KUKA KRL program: MyProgram_105().src

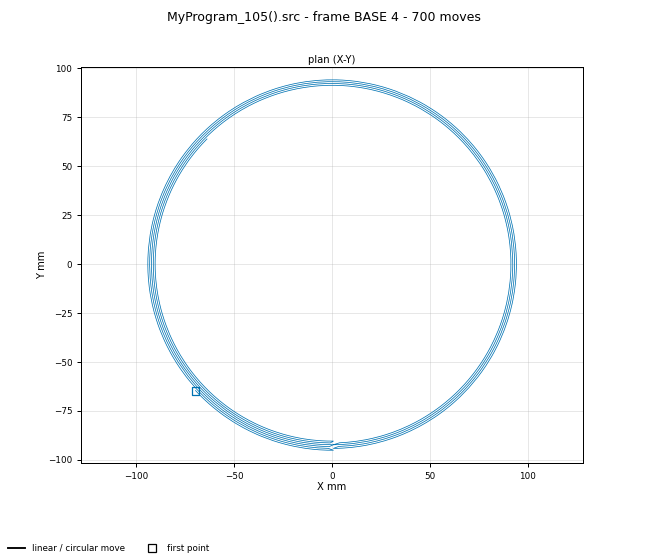
[picture p0: tool path of MyProgram_105().src in frame BASE 4, 700 of 700 moves have a stored position in this frame; points joined in program order, loops and branches not executed]
&ACCESS RVP
&REL 1
&PARAM TEMPLATE = C:\KRC\Roboter\Template\vorgabe
&PARAM EDITMASK = *
DEF MyProgram_105()
; ---- Setting reference (Base) ----
$BASE = BASE_DATA[4]

; --------------------------
; ---- Setting tool (TCP) ----
$TOOL = TOOL_DATA[3]
; --------------------------

$VEL.CP = VEL_APROX_PRINT
Startdeposition()
$VEL.CP = VEL_PRINT
LIN {X -69.7387,Y -64.5804,Z 94,A -141.1238,B 24.9322,C -1.9014,E1 24.8838,E2 -133.6356} C_DIS
LIN {X -67.3874,Y -67.0297,Z 94,A -139.0772,B 24.9325,C -1.897,E1 24.8878,E2 -135.6805} C_DIS
LIN {X -65.0404,Y -69.3086,Z 94,A -137.2267,B 24.9331,C -1.889,E1 24.8915,E2 -137.5194} C_DIS
LIN {X -62.8875,Y -71.2694,Z 94,A -135.3657,B 24.9331,C -1.889,E1 24.8954,E2 -139.3879} C_DIS
LIN {X -60.7875,Y -73.0672,Z 94,A -133.451,B 24.9327,C -1.8942,E1 24.8995,E2 -141.3222} C_DIS
LIN {X -57.6296,Y -75.5844,Z 94,A -131.3715,B 24.9339,C -1.8779,E1 24.904,E2 -143.3707} C_DIS
LIN {X -55.0629,Y -77.4728,Z 94,A -129.4404,B 24.9341,C -1.875,E1 24.9084,E2 -145.3015} C_DIS
LIN {X -51.0894,Y -80.1492,Z 94,A -126.4299,B 24.9341,C -1.8745,E1 24.9154,E2 -148.3208} C_DIS
LIN {X -49.1486,Y -81.3536,Z 94,A -124.3043,B 24.9325,C -1.898,E1 24.9207,E2 -150.5088} C_DIS
LIN {X -45.3379,Y -83.5369,Z 94,A -122.4556,B 24.9347,C -1.8671,E1 24.925,E2 -152.2894} C_DIS
LIN {X -42.3193,Y -85.1059,Z 94,A -120.7349,B 24.9356,C -1.8533,E1 24.9292,E2 -153.982} C_DIS
LIN {X -38.4134,Y -86.94,Z 94,A -117.9508,B 24.9354,C -1.8565,E1 24.9363,E2 -156.7806} C_DIS
LIN {X -36.0603,Y -87.9411,Z 94,A -116.4717,B 24.9357,C -1.8528,E1 24.9401,E2 -158.2542} C_DIS
LIN {X -30.1003,Y -90.1553,Z 94,A -112.2316,B 24.9349,C -1.8634,E1 24.9513,E2 -162.528} C_DIS
LIN {X -27.0209,Y -91.1252,Z 94,A -110.0331,B 24.9344,C -1.8708,E1 24.9573,E2 -164.7478} C_DIS
LIN {X -23.4233,Y -92.1159,Z 94,A -107.9464,B 24.9349,C -1.8638,E1 24.9629,E2 -166.8209} C_DIS
LIN {X -19.3908,Y -93.0484,Z 94,A -105.6833,B 24.9355,C -1.8545,E1 24.969,E2 -169.0649} C_DIS
LIN {X -13.8438,Y -94.0346,Z 94,A -102.1719,B 24.9353,C -1.8575,E1 24.9787,E2 -172.5866} C_DIS
LIN {X -9.7635,Y -94.5443,Z 94,A -99.8234,B 24.9357,C -1.8525,E1 24.9852,E2 -174.9249} C_DIS
LIN {X -6.5432,Y -94.8216,Z 94,A -97.8434,B 24.9356,C -1.8536,E1 24.9907,E2 -176.9083} C_DIS
LIN {X -2.4896,Y -95.0153,Z 94,A -95.2226,B 24.9351,C -1.8601,E1 24.998,E2 -179.5449} C_DIS
LIN {X 0.6469,Y -95.0437,Z 94,A -94.1191,B 24.937,C -1.8326,E1 25.0009,E2 -180.5833} C_DIS
Enddeposition()
LIN {X 0.6469,Y -95.0437,Z 94,A -94.1191,B 24.937,C -1.8326,E1 25.0009,E2 -180.5833} C_DIS
Startdeposition()
$VEL.CP = VEL_PRINT
LIN {X -1.9482,Y -94.0929,Z 94,A -96.3275,B 24.9374,C -1.8269,E1 24.9947,E2 -178.3611} C_DIS
LIN {X -6.9643,Y -93.8563,Z 94,A -99.1666,B 24.9369,C -1.8342,E1 24.9869,E2 -175.5385} C_DIS
LIN {X -11.9151,Y -93.3557,Z 94,A -101.987,B 24.9364,C -1.8417,E1 24.9791,E2 -172.7344} C_DIS
LIN {X -17.66,Y -92.4411,Z 94,A -105.2821,B 24.9358,C -1.8512,E1 24.9701,E2 -169.4586} C_DIS
LIN {X -22.5057,Y -91.3824,Z 94,A -108.5122,B 24.9362,C -1.8454,E1 24.9612,E2 -166.2106} C_DIS
LIN {X -25.5822,Y -90.5692,Z 94,A -110.5603,B 24.9363,C -1.8428,E1 24.9557,E2 -164.1533} C_DIS
LIN {X -28.6869,Y -89.6346,Z 94,A -113.2651,B 24.9379,C -1.8199,E1 24.9483,E2 -161.3892} C_DIS
LIN {X -32.4293,Y -88.3493,Z 94,A -115.1165,B 24.9365,C -1.8405,E1 24.9436,E2 -159.5831} C_DIS
LIN {X -35.4663,Y -87.1743,Z 94,A -117.1104,B 24.9364,C -1.842,E1 24.9384,E2 -157.5885} C_DIS
LIN {X -37.9827,Y -86.1086,Z 94,A -119.61,B 24.9382,C -1.8163,E1 24.9319,E2 -155.0218} C_DIS
LIN {X -42.4578,Y -83.9924,Z 94,A -121.6687,B 24.9358,C -1.8513,E1 24.9269,E2 -153.0409} C_DIS
LIN {X -48.2351,Y -80.8131,Z 94,A -125.5484,B 24.9351,C -1.8612,E1 24.9175,E2 -149.1735} C_DIS
LIN {X -50.3789,Y -79.4952,Z 94,A -128.169,B 24.9374,C -1.8282,E1 24.9111,E2 -146.4659} C_DIS
LIN {X -54.3758,Y -76.8154,Z 94,A -129.9375,B 24.9344,C -1.8706,E1 24.9072,E2 -144.7923} C_DIS
LIN {X -57.3626,Y -74.6107,Z 94,A -133.1316,B 24.9362,C -1.8443,E1 24.8999,E2 -141.5242} C_DIS
LIN {X -60.5001,Y -72.0913,Z 94,A -134.99,B 24.9346,C -1.8679,E1 24.8961,E2 -139.7148} C_DIS
LIN {X -62.7074,Y -70.1784,Z 94,A -136.6439,B 24.9341,C -1.8754,E1 24.8926,E2 -138.0722} C_DIS
LIN {X -64.8399,Y -68.2148,Z 94,A -138.555,B 24.9341,C -1.8742,E1 24.8887,E2 -136.1506} C_DIS
LIN {X -67.2732,Y -65.816,Z 94,A -140.6427,B 24.9339,C -1.8784,E1 24.8846,E2 -134.064} C_DIS
LIN {X -69.6416,Y -63.3045,Z 94,A -142.8737,B 24.9339,C -1.8789,E1 24.8803,E2 -131.8244} C_DIS
LIN {X -73.0499,Y -59.3376,Z 94,A -145.4867,B 24.932,C -1.9045,E1 24.8757,E2 -129.2603} C_DIS
LIN {X -74.6075,Y -57.3668,Z 94,A -148.2971,B 24.9346,C -1.8677,E1 24.8708,E2 -126.3489} C_DIS
LIN {X -77.3825,Y -53.5649,Z 94,A -149.7414,B 24.9309,C -1.9196,E1 24.8686,E2 -125.0212} C_DIS
LIN {X -79.2935,Y -50.6931,Z 94,A -153.1451,B 24.9335,C -1.8839,E1 24.8633,E2 -121.5154} C_DIS
LIN {X -81.4743,Y -47.1085,Z 94,A -154.6711,B 24.9307,C -1.9229,E1 24.8612,E2 -120.0743} C_DIS
LIN {X -82.5961,Y -45.113,Z 94,A -156.3966,B 24.9312,C -1.9162,E1 24.8588,E2 -118.3238} C_DIS
LIN {X -84.3717,Y -41.6972,Z 94,A -158.9654,B 24.9312,C -1.9156,E1 24.8556,E2 -115.7399} C_DIS
LIN {X -85.8006,Y -38.6713,Z 94,A -160.8303,B 24.9304,C -1.9267,E1 24.8534,E2 -113.8913} C_DIS
LIN {X -87.9215,Y -33.5723,Z 94,A -163.8897,B 24.929,C -1.9459,E1 24.8502,E2 -110.8606} C_DIS
LIN {X -88.9552,Y -30.7311,Z 94,A -166.0977,B 24.9295,C -1.9398,E1 24.8481,E2 -108.6256} C_DIS
LIN {X -89.9802,Y -27.5839,Z 94,A -168.0075,B 24.9288,C -1.9492,E1 24.8465,E2 -106.7271} C_DIS
LIN {X -90.8948,Y -24.4003,Z 94,A -170.161,B 24.9286,C -1.951,E1 24.8449,E2 -104.5656} C_DIS
LIN {X -91.8007,Y -20.7376,Z 94,A -172.5876,B 24.9284,C -1.9541,E1 24.8433,E2 -102.132} C_DIS
LIN {X -92.9269,Y -14.9027,Z 94,A -176.0707,B 24.9273,C -1.9695,E1 24.8416,E2 -98.665} C_DIS
LIN {X -93.3738,Y -11.7751,Z 94,A -178.7651,B 24.9286,C -1.952,E1 24.8406,E2 -95.9128} C_DIS
LIN {X -93.8172,Y -7.4536,Z 94,A 178.8539,B 24.9274,C -1.9684,E1 24.8401,E2 -93.5567} C_DIS
LIN {X -94.024,Y -4.0875,Z 94,A 177.0484,B 24.9263,C -1.9825,E1 24.8399,E2 -91.774} C_DIS
LIN {X -94.1117,Y -0.5106,Z 94,A 174.5652,B 24.9265,C -1.9802,E1 24.8399,E2 -89.2703} C_DIS
LIN {X -94.0669,Y 2.9403,Z 94,A 173.1792,B 24.9243,C -2.0088,E1 24.8399,E2 -87.9442} C_DIS
LIN {X -93.7885,Y 7.8127,Z 94,A 170.2835,B 24.9234,C -2.0207,E1 24.8404,E2 -85.0593} C_DIS
LIN {X -92.8908,Y 15.1219,Z 94,A 165.6955,B 24.9226,C -2.0318,E1 24.842,E2 -80.4705} C_DIS
LIN {X -91.9219,Y 20.189,Z 94,A 162.4209,B 24.9221,C -2.0376,E1 24.8438,E2 -77.1905} C_DIS
LIN {X -91.2356,Y 23.0956,Z 94,A 160.1751,B 24.9227,C -2.0303,E1 24.8453,E2 -74.914} C_DIS
LIN {X -90.0393,Y 27.3932,Z 94,A 157.4118,B 24.9222,C -2.0373,E1 24.8474,E2 -72.1515} C_DIS
LIN {X -88.776,Y 31.2417,Z 94,A 155.2063,B 24.921,C -2.053,E1 24.8494,E2 -69.9708} C_DIS
LIN {X -86.7799,Y 36.421,Z 94,A 151.5856,B 24.9207,C -2.0559,E1 24.8532,E2 -66.3368} C_DIS
LIN {X -85.0096,Y 40.3813,Z 94,A 148.9037,B 24.9202,C -2.0625,E1 24.8563,E2 -63.6561} C_DIS
LIN {X -82.7539,Y 44.822,Z 94,A 145.7368,B 24.9199,C -2.0673,E1 24.8604,E2 -60.4838} C_DIS
LIN {X -80.3279,Y 49.0375,Z 94,A 143.0972,B 24.9184,C -2.0857,E1 24.8641,E2 -57.8743} C_DIS
LIN {X -78.336,Y 52.162,Z 94,A 140.8604,B 24.9179,C -2.0926,E1 24.8675,E2 -55.6427} C_DIS
LIN {X -76.808,Y 54.3862,Z 94,A 139.1867,B 24.9176,C -2.0961,E1 24.8702,E2 -53.9692} C_DIS
LIN {X -74.738,Y 57.1974,Z 94,A 137.0233,B 24.9172,C -2.1006,E1 24.8739,E2 -51.8062} C_DIS
LIN {X -71.3643,Y 61.3558,Z 94,A 133.7903,B 24.9165,C -2.1099,E1 24.8796,E2 -48.5805} C_DIS
LIN {X -69.2025,Y 63.7831,Z 94,A 131.2365,B 24.9175,C -2.097,E1 24.8845,E2 -45.9845} C_DIS
LIN {X -66.5924,Y 66.5052,Z 94,A 128.9093,B 24.9172,C -2.1015,E1 24.8891,E2 -43.6583} C_DIS
LIN {X -63.895,Y 69.0998,Z 94,A 127.1979,B 24.9153,C -2.1246,E1 24.8925,E2 -41.9949} C_DIS
LIN {X -61.3973,Y 71.3289,Z 94,A 124.3388,B 24.917,C -2.1035,E1 24.8987,E2 -39.0743} C_DIS
LIN {X -57.8983,Y 74.195,Z 94,A 122.515,B 24.9142,C -2.1386,E1 24.9025,E2 -37.3273} C_DIS
LIN {X -55.5308,Y 75.9839,Z 94,A 120.6043,B 24.9142,C -2.139,E1 24.9068,E2 -35.4108} C_DIS
LIN {X -52.6421,Y 78.0131,Z 94,A 118.4191,B 24.9139,C -2.1421,E1 24.9118,E2 -33.2257} C_DIS
LIN {X -49.0591,Y 80.3148,Z 94,A 115.5451,B 24.9143,C -2.138,E1 24.9186,E2 -30.3328} C_DIS
LIN {X -45.2932,Y 82.4983,Z 94,A 112.9239,B 24.9138,C -2.1435,E1 24.925,E2 -27.7172} C_DIS
LIN {X -39.0636,Y 85.6239,Z 94,A 109.1301,B 24.9121,C -2.1647,E1 24.9344,E2 -23.9639} C_DIS
LIN {X -36.6843,Y 86.6689,Z 94,A 106.2784,B 24.9152,C -2.1262,E1 24.942,E2 -21.014} C_DIS
LIN {X -31.6825,Y 88.6205,Z 94,A 103.9563,B 24.9124,C -2.1609,E1 24.9479,E2 -18.7695} C_DIS
LIN {X -28.1024,Y 89.8194,Z 94,A 101.1148,B 24.9136,C -2.1459,E1 24.9555,E2 -15.8874} C_DIS
LIN {X -24.4026,Y 90.8942,Z 94,A 98.8913,B 24.9131,C -2.1523,E1 24.9615,E2 -13.6756} C_DIS
LIN {X -21.0964,Y 91.7179,Z 94,A 97.5058,B 24.9111,C -2.1768,E1 24.9651,E2 -12.3465} C_DIS
LIN {X -18.6315,Y 92.2506,Z 94,A 94.7987,B 24.9141,C -2.1396,E1 24.9728,E2 -9.5481} C_DIS
LIN {X -13.6027,Y 93.1253,Z 94,A 92.9169,B 24.9107,C -2.1821,E1 24.9777,E2 -7.7655} C_DIS
LIN {X -7.7308,Y 93.795,Z 94,A 89.1085,B 24.9111,C -2.177,E1 24.9883,E2 -3.9426} C_DIS
LIN {X -2.724,Y 94.0735,Z 94,A 86.0802,B 24.911,C -2.1789,E1 24.9967,E2 -0.918} C_DIS
LIN {X 2.2075,Y 94.0881,Z 94,A 83.1336,B 24.9108,C -2.1813,E1 25.005,E2 2.0227} C_DIS
LIN {X 5.2902,Y 93.964,Z 94,A 80.5365,B 24.9127,C -2.1571,E1 25.0124,E2 4.6762} C_DIS
LIN {X 9.0331,Y 93.6791,Z 94,A 79.1257,B 24.9103,C -2.1865,E1 25.0161,E2 6.0165} C_DIS
LIN {X 12.6316,Y 93.262,Z 94,A 76.4626,B 24.9116,C -2.1704,E1 25.0236,E2 8.7157} C_DIS
LIN {X 19.2709,Y 92.1193,Z 94,A 72.6653,B 24.9109,C -2.1793,E1 25.0339,E2 12.4877} C_DIS
LIN {X 22.378,Y 91.4136,Z 94,A 70.5662,B 24.9115,C -2.1728,E1 25.0397,E2 14.5994} C_DIS
LIN {X 25.7736,Y 90.5149,Z 94,A 67.8851,B 24.9131,C -2.1526,E1 25.047,E2 17.3237} C_DIS
LIN {X 29.3297,Y 89.4266,Z 94,A 66.1402,B 24.9118,C -2.1687,E1 25.0515,E2 19.0272} C_DIS
LIN {X 32.4829,Y 88.3297,Z 94,A 63.9325,B 24.9124,C -2.1608,E1 25.0574,E2 21.2491} C_DIS
LIN {X 39.4143,Y 85.4625,Z 94,A 59.7402,B 24.9118,C -2.169,E1 25.0681,E2 25.4121} C_DIS
LIN {X 44.9057,Y 82.7085,Z 94,A 56.0161,B 24.9121,C -2.1648,E1 25.0773,E2 29.1359} C_DIS
LIN {X 47.5693,Y 81.2066,Z 94,A 53.309,B 24.9147,C -2.1323,E1 25.084,E2 31.9119} C_DIS
LIN {X 51.1467,Y 79.0023,Z 94,A 51.6246,B 24.9126,C -2.1592,E1 25.0878,E2 33.5271} C_DIS
LIN {X 53.4154,Y 77.4865,Z 94,A 49.8003,B 24.9132,C -2.1507,E1 25.0921,E2 35.3654} C_DIS
LIN {X 55.8489,Y 75.751,Z 94,A 47.9869,B 24.9135,C -2.1478,E1 25.0962,E2 37.1794} C_DIS
LIN {X 57.8006,Y 74.2732,Z 94,A 46.327,B 24.9142,C -2.139,E1 25.0999,E2 38.8539} C_DIS
LIN {X 60.7815,Y 71.8535,Z 94,A 44.2061,B 24.9139,C -2.1423,E1 25.1044,E2 40.9588} C_DIS
LIN {X 63.4363,Y 69.5206,Z 94,A 41.9455,B 24.9146,C -2.1341,E1 25.1091,E2 43.2297} C_DIS
LIN {X 65.4276,Y 67.6496,Z 94,A 40.3764,B 24.9146,C -2.1341,E1 25.1123,E2 44.7924} C_DIS
LIN {X 69.153,Y 63.8368,Z 94,A 36.8128,B 24.9161,C -2.1155,E1 25.1192,E2 48.3845} C_DIS
LIN {X 72.2885,Y 60.2629,Z 94,A 34.2832,B 24.9155,C -2.1221,E1 25.1237,E2 50.8871} C_DIS
LIN {X 74.6663,Y 57.2905,Z 94,A 31.7816,B 24.9165,C -2.1098,E1 25.1281,E2 53.4059} C_DIS
LIN {X 76.8074,Y 54.3871,Z 94,A 29.7489,B 24.9165,C -2.1103,E1 25.1314,E2 55.4276} C_DIS
LIN {X 78.7198,Y 51.5799,Z 94,A 27.6645,B 24.9169,C -2.1044,E1 25.1346,E2 57.5155} C_DIS
LIN {X 80.6364,Y 48.53,Z 94,A 25.3599,B 24.9177,C -2.0945,E1 25.138,E2 59.8317} C_DIS
LIN {X 83.4996,Y 43.4198,Z 94,A 21.9255,B 24.9181,C -2.0897,E1 25.1426,E2 63.2596} C_DIS
LIN {X 85.0801,Y 40.2357,Z 94,A 19.7798,B 24.9185,C -2.0843,E1 25.1452,E2 65.4064} C_DIS
LIN {X 87.3911,Y 34.9333,Z 94,A 16.2834,B 24.9192,C -2.0751,E1 25.149,E2 68.9054} C_DIS
LIN {X 88.6183,Y 31.6912,Z 94,A 13.6184,B 24.9213,C -2.0484,E1 25.1516,E2 71.6186} C_DIS
LIN {X 89.8436,Y 28.0226,Z 94,A 11.6623,B 24.9207,C -2.0561,E1 25.1532,E2 73.5454} C_DIS
LIN {X 90.732,Y 25.0029,Z 94,A 9.6745,B 24.9214,C -2.0476,E1 25.1547,E2 75.5418} C_DIS
LIN {X 92.0604,Y 19.5543,Z 94,A 5.9044,B 24.9232,C -2.0238,E1 25.157,E2 79.3461} C_DIS
LIN {X 92.8381,Y 15.4375,Z 94,A 4.0615,B 24.9218,C -2.0422,E1 25.1579,E2 81.1348} C_DIS
LIN {X 93.6449,Y 9.3822,Z 94,A 0.5547,B 24.9221,C -2.0384,E1 25.1591,E2 84.6299} C_DIS
LIN {X 93.9475,Y 5.5898,Z 94,A -1.9705,B 24.9232,C -2.0232,E1 25.1596,E2 87.176} C_DIS
LIN {X 94.0861,Y 2.3126,Z 94,A -3.9319,B 24.9236,C -2.0181,E1 25.1598,E2 89.1378} C_DIS
LIN {X 94.0913,Y -2.0333,Z 94,A -6.8642,B 24.9251,C -1.9989,E1 25.1597,E2 92.098} C_DIS
LIN {X 93.8432,Y -7.1286,Z 94,A -9.5757,B 24.9247,C -2.0036,E1 25.1592,E2 94.7822} C_DIS
LIN {X 93.551,Y -10.2794,Z 94,A -12.0195,B 24.9266,C -1.978,E1 25.1585,E2 97.2719} C_DIS
LIN {X 93.103,Y -13.7597,Z 94,A -13.4432,B 24.9252,C -1.9979,E1 25.158,E2 98.6403} C_DIS
LIN {X 92.3502,Y -18.1321,Z 94,A -16.1344,B 24.9258,C -1.9896,E1 25.1567,E2 101.3353} C_DIS
LIN {X 91.8924,Y -20.3244,Z 94,A -17.7291,B 24.9268,C -1.9766,E1 25.1557,E2 102.9515} C_DIS
LIN {X 91.0157,Y -23.9512,Z 94,A -19.9981,B 24.9273,C -1.9694,E1 25.1541,E2 105.2242} C_DIS
LIN {X 89.6895,Y -28.5172,Z 94,A -22.8587,B 24.9279,C -1.9616,E1 25.1518,E2 108.0869} C_DIS
LIN {X 87.8435,Y -33.7781,Z 94,A -26.1921,B 24.9285,C -1.9534,E1 25.1487,E2 111.421} C_DIS
LIN {X 85.7242,Y -38.8408,Z 94,A -29.3311,B 24.9286,C -1.9509,E1 25.1453,E2 114.5489} C_DIS
LIN {X 84.517,Y -41.404,Z 94,A -31.2668,B 24.9296,C -1.9378,E1 25.1429,E2 116.5051} C_DIS
LIN {X 82.6594,Y -44.9962,Z 94,A -33.4527,B 24.9294,C -1.9409,E1 25.1401,E2 118.6721} C_DIS
LIN {X 81.4822,Y -47.0949,Z 94,A -35.2037,B 24.9305,C -1.9259,E1 25.1376,E2 120.4494} C_DIS
LIN {X 78.5782,Y -51.7946,Z 94,A -38.347,B 24.9305,C -1.9246,E1 25.1329,E2 123.5799} C_DIS
LIN {X 76.3889,Y -54.9736,Z 94,A -40.547,B 24.9306,C -1.9237,E1 25.1294,E2 125.7712} C_DIS
LIN {X 74.3614,Y -57.6861,Z 94,A -43.1709,B 24.9325,C -1.8972,E1 25.1249,E2 128.4451} C_DIS
LIN {X 69.8011,Y -63.1288,Z 94,A -46.9332,B 24.9318,C -1.9068,E1 25.1182,E2 132.1677} C_DIS
LIN {X 65.1773,Y -67.8909,Z 94,A -51.8243,B 24.9348,C -1.8657,E1 25.1084,E2 137.1352} C_DIS
LIN {X 62.1685,Y -70.6571,Z 94,A -53.4027,B 24.9328,C -1.8933,E1 25.1052,E2 138.6421} C_DIS
LIN {X 60.1046,Y -72.42,Z 94,A -55.9394,B 24.9353,C -1.8572,E1 25.0996,E2 141.2541} C_DIS
LIN {X 56.8954,Y -74.969,Z 94,A -58.1928,B 24.9351,C -1.8607,E1 25.0947,E2 143.4913} C_DIS
LIN {X 54.2953,Y -76.8729,Z 94,A -59.6964,B 24.9342,C -1.8733,E1 25.0913,E2 144.9597} C_DIS
LIN {X 52.3467,Y -78.2132,Z 94,A -62.078,B 24.9368,C -1.8364,E1 25.0856,E2 147.4207} C_DIS
LIN {X 48.145,Y -80.8664,Z 94,A -64.5264,B 24.9357,C -1.8515,E1 25.0799,E2 149.8258} C_DIS
LIN {X 44.3104,Y -83.0305,Z 94,A -67.7405,B 24.9374,C -1.8278,E1 25.0718,E2 153.0868} C_DIS
LIN {X 39.9429,Y -85.2164,Z 94,A -70.5367,B 24.9373,C -1.8294,E1 25.0648,E2 155.872} C_DIS
LIN {X 35.9424,Y -86.9805,Z 94,A -72.4829,B 24.9358,C -1.851,E1 25.0599,E2 157.7624} C_DIS
LIN {X 32.7951,Y -88.2157,Z 94,A -74.6569,B 24.9363,C -1.8441,E1 25.0542,E2 159.9481} C_DIS
LIN {X 30.2093,Y -89.1327,Z 94,A -76.2525,B 24.9363,C -1.8447,E1 25.05,E2 161.5392} C_DIS
LIN {X 26.5766,Y -90.2825,Z 94,A -79.3116,B 24.9382,C -1.8159,E1 25.0417,E2 164.6611} C_DIS
LIN {X 22.086,Y -91.4849,Z 94,A -80.9658,B 24.9355,C -1.8546,E1 25.0375,E2 166.2213} C_DIS
LIN {X 17.5884,Y -92.4549,Z 94,A -84.0246,B 24.9363,C -1.8429,E1 25.029,E2 169.3038} C_DIS
LIN {X 14.3248,Y -93.0162,Z 94,A -86.79,B 24.9382,C -1.8152,E1 25.0212,E2 172.1321} C_DIS
LIN {X 10.2227,Y -93.5569,Z 94,A -88.3941,B 24.9362,C -1.8456,E1 25.017,E2 173.663} C_DIS
LIN {X 5.4967,Y -93.9526,Z 94,A -91.2131,B 24.9361,C -1.8466,E1 25.0092,E2 176.4783} C_DIS
LIN {X 2.829,Y -94.0703,Z 94,A -93.0455,B 24.9366,C -1.8388,E1 25.004,E2 178.3286} C_DIS
LIN {X 0.6498,Y -94.1008,Z 94,A -94.5174,B 24.937,C -1.8335,E1 24.9998,E2 179.8128} C_DIS
Enddeposition()
LIN {X 0.6498,Y -94.1008,Z 94,A -94.5174,B 24.937,C -1.8335,E1 24.9998,E2 179.8128} C_DIS
Startdeposition()
$VEL.CP = VEL_PRINT
LIN {X 3.2914,Y -93.1215,Z 94,A -91.9183,B 24.9335,C -1.8841,E1 25.0074,E2 177.0944} C_DIS
LIN {X 10.2483,Y -92.6149,Z 94,A -87.8414,B 24.9338,C -1.8786,E1 25.0187,E2 173.0324} C_DIS
LIN {X 15.9916,Y -91.7975,Z 94,A -84.2081,B 24.9335,C -1.8834,E1 25.0288,E2 169.3912} C_DIS
LIN {X 18.5909,Y -91.3053,Z 94,A -82.0498,B 24.9321,C -1.9037,E1 25.0348,E2 167.1873} C_DIS
LIN {X 22.9029,Y -90.3203,Z 94,A -79.1877,B 24.9315,C -1.9115,E1 25.0426,E2 164.3109} C_DIS
LIN {X 26.3762,Y -89.3676,Z 94,A -77.5356,B 24.9328,C -1.8938,E1 25.0469,E2 162.7037} C_DIS
LIN {X 29.7303,Y -88.3083,Z 94,A -75.4252,B 24.9328,C -1.8945,E1 25.0525,E2 160.5955} C_DIS
LIN {X 33.1365,Y -87.0876,Z 94,A -73.0879,B 24.9322,C -1.9015,E1 25.0587,E2 158.2466} C_DIS
LIN {X 35.6068,Y -86.1085,Z 94,A -71.1636,B 24.9313,C -1.9144,E1 25.0637,E2 156.2963} C_DIS
LIN {X 39.7153,Y -84.292,Z 94,A -68.8745,B 24.9322,C -1.9014,E1 25.0694,E2 154.0435} C_DIS
LIN {X 44.1269,Y -82.0682,Z 94,A -65.6924,B 24.9315,C -1.9117,E1 25.0774,E2 150.8458} C_DIS
LIN {X 47.7244,Y -80.0298,Z 94,A -62.6462,B 24.9298,C -1.9349,E1 25.0848,E2 147.7543} C_DIS
LIN {X 50.8647,Y -78.0724,Z 94,A -60.8908,B 24.9309,C -1.9201,E1 25.0888,E2 146.0395} C_DIS
LIN {X 53.7993,Y -76.0792,Z 94,A -58.2456,B 24.9293,C -1.9417,E1 25.095,E2 143.3524} C_DIS
LIN {X 56.6324,Y -73.994,Z 94,A -56.446,B 24.93,C -1.9328,E1 25.0989,E2 141.5804} C_DIS
LIN {X 60.6404,Y -70.7465,Z 94,A -53.6631,B 24.9305,C -1.9255,E1 25.1049,E2 138.8254} C_DIS
LIN {X 63.0794,Y -68.5803,Z 94,A -51.3646,B 24.9294,C -1.9409,E1 25.1097,E2 136.4995} C_DIS
LIN {X 65.8763,Y -65.8989,Z 94,A -48.9558,B 24.9289,C -1.9477,E1 25.1145,E2 134.085} C_DIS
LIN {X 68.5042,Y -63.1624,Z 94,A -46.333,B 24.9277,C -1.9643,E1 25.1195,E2 131.4343} C_DIS
LIN {X 72.2287,Y -58.8671,Z 94,A -43.2821,B 24.9282,C -1.9568,E1 25.125,E2 128.4153} C_DIS
LIN {X 74.8639,Y -55.4791,Z 94,A -40.618,B 24.9276,C -1.9648,E1 25.1295,E2 125.7449} C_DIS
LIN {X 76.6192,Y -53.0263,Z 94,A -38.5078,B 24.9265,C -1.9795,E1 25.1329,E2 123.6102} C_DIS
LIN {X 80.2312,Y -47.3837,Z 94,A -34.8052,B 24.9268,C -1.9755,E1 25.1383,E2 119.9358} C_DIS
LIN {X 81.8823,Y -44.4695,Z 94,A -32.7879,B 24.9265,C -1.9799,E1 25.1411,E2 117.9186} C_DIS
LIN {X 83.4573,Y -41.4383,Z 94,A -30.6607,B 24.926,C -1.9872,E1 25.1438,E2 115.7856} C_DIS
LIN {X 84.7648,Y -38.6962,Z 94,A -28.1751,B 24.9238,C -2.0161,E1 25.1467,E2 113.2451} C_DIS
LIN {X 86.217,Y -35.3404,Z 94,A -26.5433,B 24.925,C -1.9996,E1 25.1484,E2 111.6612} C_DIS
LIN {X 88.2401,Y -29.9328,Z 94,A -23.0282,B 24.9243,C -2.0092,E1 25.1518,E2 108.1431} C_DIS
LIN {X 89.0893,Y -27.3028,Z 94,A -21.1469,B 24.9234,C -2.0214,E1 25.1534,E2 106.2437} C_DIS
LIN {X 90.3026,Y -22.9726,Z 94,A -18.5312,B 24.9231,C -2.0245,E1 25.1552,E2 103.6358} C_DIS
LIN {X 91.095,Y -19.5966,Z 94,A -15.3708,B 24.9196,C -2.0706,E1 25.1572,E2 100.3852} C_DIS
LIN {X 92.0816,Y -14.2557,Z 94,A -13.5788,B 24.9233,C -2.0223,E1 25.1579,E2 98.7175} C_DIS
LIN {X 92.7097,Y -9.3435,Z 94,A -10.0316,B 24.9211,C -2.051,E1 25.1592,E2 95.1236} C_DIS
LIN {X 92.9685,Y -6.2546,Z 94,A -7.5808,B 24.919,C -2.0779,E1 25.1596,E2 92.6239} C_DIS
LIN {X 93.1514,Y -2.3147,Z 94,A -5.3074,B 24.9189,C -2.0798,E1 25.1598,E2 90.3595} C_DIS
LIN {X 93.1739,Y 1.0661,Z 94,A -3.6792,B 24.9197,C -2.0694,E1 25.1598,E2 88.7656} C_DIS
LIN {X 93.0629,Y 4.6669,Z 94,A -0.9336,B 24.9176,C -2.0966,E1 25.1594,E2 85.972} C_DIS
LIN {X 92.8008,Y 8.3839,Z 94,A 0.3782,B 24.9199,C -2.0668,E1 25.1591,E2 84.7383} C_DIS
LIN {X 92.0264,Y 14.6133,Z 94,A 4.1664,B 24.9192,C -2.0762,E1 25.1578,E2 80.9503} C_DIS
LIN {X 91.485,Y 17.6848,Z 94,A 6.6821,B 24.9169,C -2.1047,E1 25.1565,E2 78.3821} C_DIS
LIN {X 90.6237,Y 21.6696,Z 94,A 9.1578,B 24.9164,C -2.1112,E1 25.1549,E2 75.9053} C_DIS
LIN {X 89.6254,Y 25.4862,Z 94,A 11.2153,B 24.9169,C -2.1048,E1 25.1535,E2 73.8748} C_DIS
LIN {X 87.5444,Y 31.9098,Z 94,A 15.4946,B 24.9156,C -2.1218,E1 25.1497,E2 69.5795} C_DIS
LIN {X 86.383,Y 34.9324,Z 94,A 17.777,B 24.9142,C -2.1385,E1 25.1473,E2 67.2703} C_DIS
LIN {X 84.2155,Y 39.8783,Z 94,A 20.6943,B 24.9147,C -2.1329,E1 25.144,E2 64.3822} C_DIS
LIN {X 81.9335,Y 44.3747,Z 94,A 24.4268,B 24.9121,C -2.165,E1 25.1391,E2 60.5936} C_DIS
LIN {X 80.1355,Y 47.5455,Z 94,A 26.1711,B 24.9131,C -2.1524,E1 25.1366,E2 58.888} C_DIS
LIN {X 78.3117,Y 50.4933,Z 94,A 28.3066,B 24.9126,C -2.1581,E1 25.1334,E2 56.7498} C_DIS
LIN {X 76.212,Y 53.6121,Z 94,A 30.3869,B 24.9129,C -2.1554,E1 25.1302,E2 54.6862} C_DIS
LIN {X 74.5248,Y 55.9313,Z 94,A 32.8088,B 24.9105,C -2.1841,E1 25.126,E2 52.2081} C_DIS
LIN {X 72.334,Y 58.7371,Z 94,A 34.5233,B 24.9115,C -2.1717,E1 25.1231,E2 50.5308} C_DIS
LIN {X 70.0892,Y 61.3985,Z 94,A 37.4122,B 24.9089,C -2.2042,E1 25.1177,E2 47.578} C_DIS
LIN {X 66.9704,Y 64.7862,Z 94,A 39.4361,B 24.9108,C -2.1806,E1 25.1139,E2 45.6187} C_DIS
LIN {X 64.5539,Y 67.1943,Z 94,A 41.456,B 24.9107,C -2.1822,E1 25.1099,E2 43.6035} C_DIS
LIN {X 60.9408,Y 70.489,Z 94,A 44.5547,B 24.9099,C -2.1915,E1 25.1034,E2 40.4952} C_DIS
LIN {X 59.052,Y 72.0788,Z 94,A 46.125,B 24.9095,C -2.1962,E1 25.1,E2 38.9197} C_DIS
LIN {X 56.5971,Y 74.0213,Z 94,A 48.1948,B 24.9088,C -2.205,E1 25.0954,E2 36.8369} C_DIS
LIN {X 52.9441,Y 76.6763,Z 94,A 50.6792,B 24.9093,C -2.1991,E1 25.0898,E2 34.3749} C_DIS
LIN {X 48.4077,Y 79.6174,Z 94,A 54.0116,B 24.9088,C -2.2045,E1 25.0819,E2 31.0405} C_DIS
LIN {X 45.3335,Y 81.4072,Z 94,A 55.8988,B 24.9095,C -2.197,E1 25.0774,E2 29.1769} C_DIS
LIN {X 39.8714,Y 84.2188,Z 94,A 59.9732,B 24.9082,C -2.2122,E1 25.0672,E2 25.0775} C_DIS
LIN {X 34.5103,Y 86.5536,Z 94,A 63.6897,B 24.9075,C -2.2203,E1 25.0576,E2 21.3506} C_DIS
LIN {X 30.9656,Y 87.8829,Z 94,A 65.6061,B 24.9086,C -2.208,E1 25.0527,E2 19.4674} C_DIS
LIN {X 26.0415,Y 89.4669,Z 94,A 69.0272,B 24.9077,C -2.2188,E1 25.0435,E2 16.0269} C_DIS
LIN {X 23.0761,Y 90.276,Z 94,A 70.857,B 24.9077,C -2.2179,E1 25.0386,E2 14.2021} C_DIS
LIN {X 20.7277,Y 90.8442,Z 94,A 72.5671,B 24.907,C -2.2264,E1 25.0339,E2 12.474} C_DIS
LIN {X 15.1554,Y 91.9381,Z 94,A 75.9548,B 24.9072,C -2.2242,E1 25.0246,E2 9.0955} C_DIS
LIN {X 8.6612,Y 92.7752,Z 94,A 79.575,B 24.9083,C -2.211,E1 25.0147,E2 5.5093} C_DIS
LIN {X 3.6923,Y 93.1059,Z 94,A 82.8341,B 24.9077,C -2.2176,E1 25.0056,E2 2.2358} C_DIS
LIN {X -2.0956,Y 93.1558,Z 94,A 86.7375,B 24.9068,C -2.2286,E1 24.9946,E2 -1.6934} C_DIS
LIN {X -7.6443,Y 92.8648,Z 94,A 89.6946,B 24.9082,C -2.2118,E1 24.9865,E2 -4.6116} C_DIS
LIN {X -13.835,Y 92.1467,Z 94,A 93.5529,B 24.9084,C -2.2103,E1 24.9758,E2 -8.4691} C_DIS
LIN {X -19.2391,Y 91.1722,Z 94,A 97.2689,B 24.9076,C -2.2189,E1 24.9655,E2 -12.2094} C_DIS
LIN {X -21.8619,Y 90.5779,Z 94,A 99.7551,B 24.9054,C -2.2451,E1 24.9586,E2 -14.7614} C_DIS
LIN {X -26.5767,Y 89.3081,Z 94,A 101.8119,B 24.9083,C -2.2104,E1 24.9533,E2 -16.7391} C_DIS
LIN {X -29.7671,Y 88.2959,Z 94,A 103.6106,B 24.9093,C -2.1995,E1 24.9485,E2 -18.5151} C_DIS
LIN {X -33.957,Y 86.7709,Z 94,A 107.2306,B 24.9072,C -2.2247,E1 24.9389,E2 -22.2025} C_DIS
LIN {X -37.3474,Y 85.3665,Z 94,A 108.8945,B 24.909,C -2.202,E1 24.9348,E2 -23.8164} C_DIS
LIN {X -42.6543,Y 82.8429,Z 94,A 112.9932,B 24.9082,C -2.212,E1 24.9244,E2 -27.9497} C_DIS
LIN {X -46.7524,Y 80.6015,Z 94,A 115.487,B 24.9096,C -2.1947,E1 24.9184,E2 -30.4095} C_DIS
LIN {X -49.8777,Y 78.7068,Z 94,A 117.8468,B 24.9096,C -2.1941,E1 24.9128,E2 -32.7754} C_DIS
LIN {X -53.2048,Y 76.4951,Z 94,A 120.1566,B 24.9105,C -2.1846,E1 24.9075,E2 -35.0703} C_DIS
LIN {X -56.1183,Y 74.3843,Z 94,A 123.3638,B 24.9082,C -2.2121,E1 24.9002,E2 -38.3544} C_DIS
LIN {X -60.1304,Y 71.181,Z 94,A 125.5502,B 24.9114,C -2.1739,E1 24.8957,E2 -40.4582} C_DIS
LIN {X -62.598,Y 69.022,Z 94,A 127.6474,B 24.9115,C -2.1719,E1 24.8913,E2 -42.5589} C_DIS
LIN {X -66.1153,Y 65.6588,Z 94,A 130.9478,B 24.9113,C -2.1745,E1 24.8847,E2 -45.8795} C_DIS
LIN {X -69.3234,Y 62.2619,Z 94,A 133.4609,B 24.9128,C -2.156,E1 24.88,E2 -48.3594} C_DIS
LIN {X -71.3342,Y 59.9495,Z 94,A 136.0473,B 24.9114,C -2.1733,E1 24.8753,E2 -50.999} C_DIS
LIN {X -73.8181,Y 56.8608,Z 94,A 137.7695,B 24.9138,C -2.1443,E1 24.8724,E2 -52.6601} C_DIS
LIN {X -75.8326,Y 54.1449,Z 94,A 139.8967,B 24.9141,C -2.1402,E1 24.8689,E2 -54.7878} C_DIS
LIN {X -77.3263,Y 51.9902,Z 94,A 141.6584,B 24.9141,C -2.1404,E1 24.8661,E2 -56.5588} C_DIS
LIN {X -79.3802,Y 48.7982,Z 94,A 143.9166,B 24.9148,C -2.1314,E1 24.8628,E2 -58.807} C_DIS
LIN {X -82.2505,Y 43.7868,Z 94,A 147.4953,B 24.9156,C -2.122,E1 24.8579,E2 -62.382} C_DIS
LIN {X -84.6675,Y 38.9085,Z 94,A 150.8241,B 24.9164,C -2.1114,E1 24.8539,E2 -65.7037} C_DIS
LIN {X -85.7078,Y 36.5595,Z 94,A 153.2367,B 24.9147,C -2.1326,E1 24.8512,E2 -68.1802} C_DIS
LIN {X -87.3826,Y 32.3533,Z 94,A 155.2484,B 24.9173,C -2.1,E1 24.8493,E2 -70.1253} C_DIS
LIN {X -88.3047,Y 29.7411,Z 94,A 157.1625,B 24.9172,C -2.1012,E1 24.8475,E2 -72.0534} C_DIS
LIN {X -89.6428,Y 25.4247,Z 94,A 159.7005,B 24.9185,C -2.0851,E1 24.8455,E2 -74.5674} C_DIS
LIN {X -90.5207,Y 22.0964,Z 94,A 161.7975,B 24.919,C -2.0778,E1 24.8441,E2 -76.6593} C_DIS
LIN {X -91.1619,Y 19.2891,Z 94,A 164.2361,B 24.9179,C -2.0929,E1 24.8426,E2 -79.1482} C_DIS
LIN {X -91.8473,Y 15.6985,Z 94,A 165.6303,B 24.9205,C -2.0593,E1 24.842,E2 -80.4705} C_DIS
LIN {X -92.5284,Y 10.9893,Z 94,A 168.8462,B 24.9205,C -2.0588,E1 24.8408,E2 -83.7044} C_DIS
LIN {X -92.8693,Y 7.5875,Z 94,A 170.8247,B 24.9213,C -2.0482,E1 24.8402,E2 -85.6696} C_DIS
LIN {X -93.1159,Y 3.4561,Z 94,A 174.3057,B 24.9197,C -2.0691,E1 24.8398,E2 -89.2214} C_DIS
LIN {X -93.1755,Y -0.8477,Z 94,A 176.0725,B 24.9225,C -2.0333,E1 24.8398,E2 -90.9133} C_DIS
LIN {X -92.9273,Y -6.8625,Z 94,A 179.782,B 24.9234,C -2.0216,E1 24.8403,E2 -94.6173} C_DIS
LIN {X -92.5083,Y -11.1615,Z 94,A -177.362,B 24.9235,C -2.0194,E1 24.8411,E2 -97.4852} C_DIS
LIN {X -92.0422,Y -14.5106,Z 94,A -175.3181,B 24.9241,C -2.0118,E1 24.842,E2 -99.523} C_DIS
LIN {X -91.1752,Y -19.224,Z 94,A -172.2501,B 24.9245,C -2.0064,E1 24.8436,E2 -102.5962} C_DIS
LIN {X -90.4415,Y -22.421,Z 94,A -170.2426,B 24.925,C -1.9999,E1 24.8449,E2 -104.6001} C_DIS
LIN {X -89.5464,Y -25.7651,Z 94,A -168.1255,B 24.9255,C -1.9931,E1 24.8465,E2 -106.7132} C_DIS
LIN {X -88.5253,Y -29.0808,Z 94,A -166.1584,B 24.9264,C -1.9815,E1 24.8481,E2 -108.664} C_DIS
LIN {X -87.8315,Y -31.112,Z 94,A -164.5745,B 24.9261,C -1.9859,E1 24.8496,E2 -110.2673} C_DIS
LIN {X -86.3446,Y -35.0267,Z 94,A -161.7799,B 24.9261,C -1.9853,E1 24.8525,E2 -113.0762} C_DIS
LIN {X -84.5217,Y -39.2217,Z 94,A -159.4756,B 24.9279,C -1.9614,E1 24.8551,E2 -115.336} C_DIS
LIN {X -82.5612,Y -43.1969,Z 94,A -156.5373,B 24.9279,C -1.9605,E1 24.8588,E2 -118.288} C_DIS
LIN {X -80.9968,Y -46.0646,Z 94,A -154.7322,B 24.9288,C -1.9486,E1 24.8612,E2 -120.0743} C_DIS
LIN {X -78.4931,Y -50.2106,Z 94,A -151.3534,B 24.9285,C -1.9535,E1 24.8662,E2 -123.4821} C_DIS
LIN {X -73.5996,Y -57.1443,Z 94,A -146.2415,B 24.9296,C -1.9371,E1 24.8745,E2 -128.5798} C_DIS
LIN {X -70.1694,Y -61.3067,Z 94,A -142.9473,B 24.9303,C -1.9287,E1 24.8804,E2 -131.8691} C_DIS
LIN {X -67.857,Y -63.8567,Z 94,A -140.8395,B 24.9306,C -1.9238,E1 24.8844,E2 -133.9743} C_DIS
LIN {X -65.4928,Y -66.2793,Z 94,A -138.7695,B 24.931,C -1.919,E1 24.8885,E2 -136.0417} C_DIS
LIN {X -63.1472,Y -68.518,Z 94,A -136.6394,B 24.931,C -1.9193,E1 24.8928,E2 -138.1814} C_DIS
LIN {X -60.2117,Y -71.1118,Z 94,A -133.1597,B 24.9287,C -1.9499,E1 24.9004,E2 -141.7474} C_DIS
LIN {X -55.862,Y -74.5768,Z 94,A -130.9791,B 24.9321,C -1.903,E1 24.905,E2 -143.8242} C_DIS
LIN {X -52.1729,Y -77.2027,Z 94,A -127.635,B 24.9311,C -1.9168,E1 24.9128,E2 -147.2126} C_DIS
LIN {X -48.2625,Y -79.7058,Z 94,A -125.3392,B 24.9327,C -1.894,E1 24.9181,E2 -149.4614} C_DIS
LIN {X -43.0441,Y -82.6416,Z 94,A -121.4825,B 24.9327,C -1.8948,E1 24.9276,E2 -153.3309} C_DIS
LIN {X -40.6817,Y -83.8295,Z 94,A -119.3485,B 24.9316,C -1.9098,E1 24.9331,E2 -155.5063} C_DIS
LIN {X -37.552,Y -85.2773,Z 94,A -117.5842,B 24.9326,C -1.8955,E1 24.9375,E2 -157.2409} C_DIS
LIN {X -33.9039,Y -86.7918,Z 94,A -115.6356,B 24.934,C -1.877,E1 24.9424,E2 -159.1498} C_DIS
LIN {X -29.3053,Y -88.4517,Z 94,A -112.2664,B 24.9333,C -1.8866,E1 24.9514,E2 -162.5484} C_DIS
LIN {X -26.0544,Y -89.463,Z 94,A -110.1257,B 24.9333,C -1.8867,E1 24.9571,E2 -164.693} C_DIS
LIN {X -21.768,Y -90.6008,Z 94,A -106.8808,B 24.9321,C -1.903,E1 24.966,E2 -167.981} C_DIS
LIN {X -18.1192,Y -91.4014,Z 94,A -105.113,B 24.9335,C -1.8838,E1 24.9707,E2 -169.7053} C_DIS
LIN {X -14.0135,Y -92.1191,Z 94,A -102.4496,B 24.9333,C -1.8865,E1 24.9781,E2 -172.3777} C_DIS
LIN {X -7.6203,Y -92.8667,Z 94,A -98.6745,B 24.9338,C -1.8797,E1 24.9885,E2 -176.1389} C_DIS
LIN {X -5.0764,Y -93.0402,Z 94,A -96.503,B 24.9323,C -1.9008,E1 24.9947,E2 -178.3612} C_DIS
LIN {X -1.4057,Y -93.1685,Z 94,A -93.9531,B 24.9315,C -1.9115,E1 25.0019,E2 -180.9365} C_DIS
LIN {X -1.4057,Y -93.1685,Z 94,A -93.9531,B 24.9315,C -1.9115,E1 25.0019,E2 -180.9365} C_DIS
Enddeposition()
LIN {X 0.6403,Y -92.241,Z 94,A -94.4274,B 24.9346,C -1.8679,E1 25.0003,E2 -180.3586} C_DIS
Startdeposition()
$VEL.CP = VEL_PRINT
LIN {X -5.4551,Y -92.0837,Z 94,A -98.1404,B 24.9345,C -1.8698,E1 24.99,E2 -176.6497} C_DIS
LIN {X -9.6737,Y -91.7358,Z 94,A -100.9603,B 24.9349,C -1.8636,E1 24.9821,E2 -173.8136} C_DIS
LIN {X -14.6853,Y -91.0695,Z 94,A -103.9212,B 24.9344,C -1.8702,E1 24.9739,E2 -170.8661} C_DIS
LIN {X -17.1169,Y -90.643,Z 94,A -105.5917,B 24.9347,C -1.8662,E1 24.9693,E2 -169.1843} C_DIS
LIN {X -21.0274,Y -89.8162,Z 94,A -108.0991,B 24.9347,C -1.8665,E1 24.9625,E2 -166.6746} C_DIS
LIN {X -23.4635,Y -89.2119,Z 94,A -109.7752,B 24.9349,C -1.8636,E1 24.9579,E2 -164.9889} C_DIS
LIN {X -26.9203,Y -88.2298,Z 94,A -111.8822,B 24.9345,C -1.8692,E1 24.9523,E2 -162.8919} C_DIS
LIN {X -29.6817,Y -87.3389,Z 94,A -114.0532,B 24.9352,C -1.8586,E1 24.9465,E2 -160.6917} C_DIS
LIN {X -33.9357,Y -85.7756,Z 94,A -116.7043,B 24.9347,C -1.8666,E1 24.9396,E2 -158.0538} C_DIS
LIN {X -36.885,Y -84.549,Z 94,A -118.6667,B 24.9345,C -1.8694,E1 24.9345,E2 -156.0936} C_DIS
LIN {X -40.1192,Y -83.0633,Z 94,A -120.7361,B 24.934,C -1.8765,E1 24.9293,E2 -154.0359} C_DIS
LIN {X -43.4315,Y -81.3818,Z 94,A -123.5549,B 24.9349,C -1.8631,E1 24.9223,E2 -151.1773} C_DIS
LIN {X -46.3995,Y -79.7269,Z 94,A -125.0185,B 24.9333,C -1.8867,E1 24.9189,E2 -149.7656} C_DIS
LIN {X -48.8455,Y -78.2506,Z 94,A -128.246,B 24.9363,C -1.8435,E1 24.911,E2 -146.4251} C_DIS
LIN {X -53.9752,Y -74.8061,Z 94,A -130.6054,B 24.9326,C -1.8963,E1 24.9059,E2 -144.1833} C_DIS
LIN {X -59.9227,Y -70.1307,Z 94,A -135.4052,B 24.9322,C -1.9017,E1 24.8953,E2 -139.3785} C_DIS
LIN {X -62.028,Y -68.2772,Z 94,A -137.3614,B 24.9324,C -1.8984,E1 24.8912,E2 -137.4065} C_DIS
LIN {X -64.6496,Y -65.7991,Z 94,A -139.5328,B 24.932,C -1.9052,E1 24.8869,E2 -135.2423} C_DIS
LIN {X -67.0104,Y -63.3933,Z 94,A -141.6028,B 24.9316,C -1.9104,E1 24.8829,E2 -133.1759} C_DIS
LIN {X -69.2653,Y -60.9217,Z 94,A -143.7073,B 24.9313,C -1.9142,E1 24.879,E2 -131.0711} C_DIS
LIN {X -71.8044,Y -57.9069,Z 94,A -146.0439,B 24.9306,C -1.9234,E1 24.8748,E2 -128.7456} C_DIS
LIN {X -75.4331,Y -53.0959,Z 94,A -149.9944,B 24.9305,C -1.9261,E1 24.8682,E2 -124.7824} C_DIS
LIN {X -77.2515,Y -50.4125,Z 94,A -152.766,B 24.9317,C -1.9081,E1 24.8639,E2 -121.9541} C_DIS
LIN {X -79.5698,Y -46.6667,Z 94,A -154.5361,B 24.9291,C -1.9448,E1 24.8615,E2 -120.2623} C_DIS
LIN {X -80.8806,Y -44.357,Z 94,A -156.3977,B 24.9292,C -1.9427,E1 24.8589,E2 -118.386} C_DIS
LIN {X -82.7927,Y -40.6757,Z 94,A -158.7596,B 24.9282,C -1.9564,E1 24.8559,E2 -116.044} C_DIS
LIN {X -83.917,Y -38.3037,Z 94,A -160.6006,B 24.9284,C -1.9545,E1 24.8538,E2 -114.1886} C_DIS
LIN {X -86.136,Y -33.0115,Z 94,A -163.928,B 24.9271,C -1.972,E1 24.8503,E2 -110.8843} C_DIS
LIN {X -87.3858,Y -29.5426,Z 94,A -166.0646,B 24.9262,C -1.9834,E1 24.8482,E2 -108.7629} C_DIS
LIN {X -88.5058,Y -25.9965,Z 94,A -168.8124,B 24.9267,C -1.977,E1 24.8459,E2 -105.9841} C_DIS
LIN {X -89.4071,Y -22.704,Z 94,A -170.934,B 24.9262,C -1.9835,E1 24.8444,E2 -103.8654} C_DIS
LIN {X -90.1719,Y -19.445,Z 94,A -173.1432,B 24.9261,C -1.986,E1 24.8431,E2 -101.6491} C_DIS
LIN {X -90.8971,Y -15.7167,Z 94,A -175.5155,B 24.9255,C -1.9929,E1 24.8419,E2 -99.2794} C_DIS
LIN {X -91.4489,Y -12.0912,Z 94,A -177.74,B 24.9249,C -2.0017,E1 24.841,E2 -97.0626} C_DIS
LIN {X -91.9186,Y -7.7568,Z 94,A 179.6488,B 24.924,C -2.0131,E1 24.8403,E2 -94.463} C_DIS
LIN {X -92.1889,Y -3.223,Z 94,A 176.7424,B 24.9235,C -2.0196,E1 24.8398,E2 -91.5545} C_DIS
LIN {X -92.2455,Y -0.0816,Z 94,A 174.301,B 24.9242,C -2.0112,E1 24.8398,E2 -89.0784} C_DIS
LIN {X -92.1044,Y 5.08,Z 94,A 171.5319,B 24.9224,C -2.0346,E1 24.8401,E2 -86.3485} C_DIS
LIN {X -91.8567,Y 8.4484,Z 94,A 169.3919,B 24.922,C -2.04,E1 24.8406,E2 -84.2087} C_DIS
LIN {X -91.4605,Y 12.0011,Z 94,A 166.8615,B 24.9221,C -2.0379,E1 24.8415,E2 -81.658} C_DIS
LIN {X -90.867,Y 15.888,Z 94,A 164.4276,B 24.9215,C -2.0459,E1 24.8426,E2 -79.2289} C_DIS
LIN {X -90.1424,Y 19.5802,Z 94,A 162.3666,B 24.9203,C -2.0616,E1 24.8437,E2 -77.1931} C_DIS
LIN {X -89.329,Y 23.0081,Z 94,A 160.2169,B 24.9197,C -2.0697,E1 24.8452,E2 -75.0501} C_DIS
LIN {X -88.5103,Y 25.9815,Z 94,A 157.541,B 24.921,C -2.0531,E1 24.8473,E2 -72.3191} C_DIS
LIN {X -87.3031,Y 29.7877,Z 94,A 155.6476,B 24.919,C -2.0782,E1 24.8489,E2 -70.4748} C_DIS
LIN {X -85.5086,Y 34.6027,Z 94,A 152.7188,B 24.9176,C -2.0959,E1 24.8518,E2 -67.5717} C_DIS
LIN {X -84.3659,Y 37.3049,Z 94,A 150.6129,B 24.9179,C -2.0928,E1 24.8542,E2 -65.4469} C_DIS
LIN {X -81.9398,Y 42.3681,Z 94,A 147.3378,B 24.9165,C -2.1096,E1 24.8582,E2 -62.1941} C_DIS
LIN {X -80.892,Y 44.3361,Z 94,A 145.2658,B 24.9179,C -2.093,E1 24.861,E2 -60.0715} C_DIS
LIN {X -79.2152,Y 47.2667,Z 94,A 143.8105,B 24.9158,C -2.1182,E1 24.863,E2 -58.669} C_DIS
LIN {X -77.624,Y 49.8351,Z 94,A 141.7184,B 24.9159,C -2.117,E1 24.8661,E2 -56.5633} C_DIS
LIN {X -75.8362,Y 52.516,Z 94,A 139.7847,B 24.9153,C -2.1246,E1 24.8691,E2 -54.6381} C_DIS
LIN {X -73.9938,Y 55.0828,Z 94,A 137.7524,B 24.9151,C -2.1278,E1 24.8725,E2 -52.6036} C_DIS
LIN {X -71.3037,Y 58.5244,Z 94,A 135.2089,B 24.9141,C -2.1401,E1 24.8769,E2 -50.0775} C_DIS
LIN {X -69.4653,Y 60.6927,Z 94,A 133.3214,B 24.9141,C -2.1409,E1 24.8803,E2 -48.1833} C_DIS
LIN {X -67.1446,Y 63.2507,Z 94,A 130.967,B 24.9141,C -2.1399,E1 24.8848,E2 -45.8161} C_DIS
LIN {X -64.0427,Y 66.3895,Z 94,A 128.4022,B 24.9132,C -2.1518,E1 24.8899,E2 -43.2689} C_DIS
LIN {X -61.5893,Y 68.6716,Z 94,A 126.2879,B 24.9128,C -2.1556,E1 24.8942,E2 -41.1551} C_DIS
LIN {X -58.9559,Y 70.9453,Z 94,A 123.5558,B 24.9139,C -2.1429,E1 24.9001,E2 -38.3823} C_DIS
LIN {X -56.1978,Y 73.1496,Z 94,A 122.0931,B 24.9117,C -2.17,E1 24.9032,E2 -36.9788} C_DIS
LIN {X -54.0134,Y 74.7788,Z 94,A 120.1208,B 24.9121,C -2.1648,E1 24.9077,E2 -34.9871} C_DIS
LIN {X -51.1173,Y 76.7869,Z 94,A 117.9077,B 24.9118,C -2.1684,E1 24.9128,E2 -32.7751} C_DIS
LIN {X -48.7849,Y 78.2884,Z 94,A 116.3512,B 24.9111,C -2.1768,E1 24.9165,E2 -31.2337} C_DIS
LIN {X -46.4978,Y 79.6696,Z 94,A 114.7549,B 24.9107,C -2.1817,E1 24.9203,E2 -29.6444} C_DIS
LIN {X -42.1928,Y 82.0296,Z 94,A 111.6309,B 24.9105,C -2.1846,E1 24.928,E2 -26.5182} C_DIS
LIN {X -39.5593,Y 83.3324,Z 94,A 109.6422,B 24.9107,C -2.1823,E1 24.933,E2 -24.519} C_DIS
LIN {X -36.5791,Y 84.6823,Z 94,A 107.6768,B 24.9103,C -2.1874,E1 24.938,E2 -22.5609} C_DIS
LIN {X -30.5744,Y 87.0301,Z 94,A 103.8111,B 24.9095,C -2.1971,E1 24.948,E2 -18.7102} C_DIS
LIN {X -27.866,Y 87.9365,Z 94,A 101.1274,B 24.9117,C -2.1703,E1 24.9554,E2 -15.958} C_DIS
LIN {X -23.8665,Y 89.1037,Z 94,A 99.5025,B 24.9089,C -2.2036,E1 24.9595,E2 -14.4099} C_DIS
LIN {X -21.5054,Y 89.7033,Z 94,A 97.7876,B 24.9093,C -2.1986,E1 24.9642,E2 -12.6805} C_DIS
LIN {X -18.3169,Y 90.4079,Z 94,A 95.2459,B 24.9105,C -2.1838,E1 24.9713,E2 -10.1008} C_DIS
LIN {X -15.0508,Y 91.0084,Z 94,A 93.854,B 24.9086,C -2.207,E1 24.9749,E2 -8.7625} C_DIS
LIN {X -10.2553,Y 91.6738,Z 94,A 90.7594,B 24.9087,C -2.2059,E1 24.9835,E2 -5.6631} C_DIS
LIN {X -7.1027,Y 91.9709,Z 94,A 88.1015,B 24.9105,C -2.1844,E1 24.9911,E2 -2.9529} C_DIS
LIN {X -3.4352,Y 92.1808,Z 94,A 86.5589,B 24.9084,C -2.2093,E1 24.9952,E2 -1.469} C_DIS
LIN {X 2.0466,Y 92.2224,Z 94,A 83.2393,B 24.9082,C -2.2128,E1 25.0045,E2 1.8423} C_DIS
LIN {X 7.1606,Y 91.9663,Z 94,A 79.8674,B 24.9087,C -2.2064,E1 25.0139,E2 5.2279} C_DIS
LIN {X 11.6,Y 91.5125,Z 94,A 77.3697,B 24.908,C -2.2152,E1 25.0208,E2 7.7032} C_DIS
LIN {X 14.02,Y 91.1728,Z 94,A 75.5539,B 24.9088,C -2.2048,E1 25.0258,E2 9.542} C_DIS
LIN {X 17.7804,Y 90.5153,Z 94,A 73.1467,B 24.909,C -2.2026,E1 25.0325,E2 11.9516} C_DIS
LIN {X 20.2489,Y 89.9958,Z 94,A 71.6175,B 24.909,C -2.2031,E1 25.0366,E2 13.4776} C_DIS
LIN {X 23.2363,Y 89.2703,Z 94,A 69.6176,B 24.9093,C -2.1989,E1 25.0421,E2 15.4844} C_DIS
LIN {X 26.5988,Y 88.3271,Z 94,A 67.2114,B 24.9101,C -2.1894,E1 25.0486,E2 17.9091} C_DIS
LIN {X 30.7634,Y 86.9638,Z 94,A 64.6182,B 24.9099,C -2.1914,E1 25.0554,E2 20.4924} C_DIS
LIN {X 33.9246,Y 85.78,Z 94,A 62.3963,B 24.9104,C -2.1851,E1 25.0612,E2 22.7243} C_DIS
LIN {X 37.2905,Y 84.3722,Z 94,A 60.4203,B 24.9098,C -2.1925,E1 25.0662,E2 24.678} C_DIS
LIN {X 40.4902,Y 82.8846,Z 94,A 57.7345,B 24.9114,C -2.1729,E1 25.073,E2 27.4032} C_DIS
LIN {X 43.5739,Y 81.3054,Z 94,A 56.1785,B 24.91,C -2.1906,E1 25.0768,E2 28.913} C_DIS
LIN {X 46.1489,Y 79.8709,Z 94,A 53.2137,B 24.9134,C -2.149,E1 25.0842,E2 31.9673} C_DIS
LIN {X 50.7324,Y 77.0405,Z 94,A 51.0217,B 24.9106,C -2.1836,E1 25.0891,E2 34.0704} C_DIS
LIN {X 52.8633,Y 75.5948,Z 94,A 48.7379,B 24.9127,C -2.1571,E1 25.0944,E2 36.409} C_DIS
LIN {X 55.9732,Y 73.3227,Z 94,A 46.9148,B 24.9115,C -2.1726,E1 25.0984,E2 38.1886} C_DIS
LIN {X 58.7963,Y 71.0779,Z 94,A 44.7812,B 24.9115,C -2.1722,E1 25.103,E2 40.3152} C_DIS
LIN {X 61.6673,Y 68.6018,Z 94,A 42.6151,B 24.9113,C -2.1743,E1 25.1076,E2 42.4679} C_DIS
LIN {X 63.5117,Y 66.899,Z 94,A 40.789,B 24.9124,C -2.1616,E1 25.1113,E2 44.3164} C_DIS
LIN {X 65.8983,Y 64.5492,Z 94,A 38.7393,B 24.9126,C -2.1583,E1 25.1154,E2 46.3653} C_DIS
LIN {X 69.2649,Y 60.9222,Z 94,A 35.7236,B 24.913,C -2.1535,E1 25.121,E2 49.379} C_DIS
LIN {X 71.4583,Y 58.3339,Z 94,A 32.7218,B 24.916,C -2.1168,E1 25.1265,E2 52.4535} C_DIS
LIN {X 74.3816,Y 54.5565,Z 94,A 30.9098,B 24.9132,C -2.1507,E1 25.1294,E2 54.1769} C_DIS
LIN {X 75.8558,Y 52.4878,Z 94,A 29.0975,B 24.9142,C -2.1383,E1 25.1323,E2 56.0096} C_DIS
LIN {X 77.6799,Y 49.7482,Z 94,A 27.1403,B 24.9144,C -2.1362,E1 25.1353,E2 57.9621} C_DIS
LIN {X 79.4488,Y 46.8713,Z 94,A 24.5024,B 24.9164,C -2.1112,E1 25.1391,E2 60.6454} C_DIS
LIN {X 81.0902,Y 43.9707,Z 94,A 22.4658,B 24.9168,C -2.1068,E1 25.1418,E2 62.6818} C_DIS
LIN {X 82.5953,Y 41.074,Z 94,A 21.315,B 24.9147,C -2.1329,E1 25.1432,E2 63.7648} C_DIS
LIN {X 83.6224,Y 38.9402,Z 94,A 18.5782,B 24.9186,C -2.083,E1 25.1466,E2 66.6047} C_DIS
LIN {X 85.497,Y 34.6312,Z 94,A 16.4942,B 24.9169,C -2.1046,E1 25.1487,E2 68.626} C_DIS
LIN {X 86.7781,Y 31.2844,Z 94,A 13.6692,B 24.9191,C -2.0764,E1 25.1515,E2 71.5019} C_DIS
LIN {X 88.0422,Y 27.5254,Z 94,A 12.0203,B 24.9174,C -2.0986,E1 25.1528,E2 73.0891} C_DIS
LIN {X 88.8096,Y 24.9386,Z 94,A 10.1457,B 24.9184,C -2.0863,E1 25.1543,E2 74.9821} C_DIS
LIN {X 89.9649,Y 20.3839,Z 94,A 6.6796,B 24.9206,C -2.0574,E1 25.1566,E2 78.4962} C_DIS
LIN {X 90.743,Y 16.5773,Z 94,A 5.2545,B 24.9184,C -2.086,E1 25.1573,E2 79.8455} C_DIS
LIN {X 91.1654,Y 14.0675,Z 94,A 2.8863,B 24.921,C -2.0522,E1 25.1583,E2 82.2797} C_DIS
LIN {X 91.6105,Y 10.7959,Z 94,A 1.1375,B 24.9207,C -2.0567,E1 25.1589,E2 84.0074} C_DIS
LIN {X 92.1691,Y 3.7343,Z 94,A -2.4483,B 24.9194,C -2.0727,E1 25.1597,E2 87.5341} C_DIS
LIN {X 92.2411,Y -0.806,Z 94,A -5.8863,B 24.9219,C -2.0408,E1 25.1597,E2 91.0269} C_DIS
LIN {X 92.1205,Y -4.7669,Z 94,A -8.6117,B 24.9232,C -2.0232,E1 25.1594,E2 93.7777} C_DIS
LIN {X 91.8761,Y -8.2382,Z 94,A -11.6992,B 24.9263,C -1.9825,E1 25.1586,E2 96.9428} C_DIS
LIN {X 91.1389,Y -14.2395,Z 94,A -15.0596,B 24.9261,C -1.9848,E1 25.1572,E2 100.2781} C_DIS
LIN {X 90.2773,Y -18.9529,Z 94,A -17.1579,B 24.9244,C -2.0074,E1 25.1561,E2 102.311} C_DIS
LIN {X 88.8627,Y -24.7513,Z 94,A -20.7882,B 24.9251,C -1.9984,E1 25.1536,E2 105.9414} C_DIS
LIN {X 87.9235,Y -27.9062,Z 94,A -22.9319,B 24.9259,C -1.9884,E1 25.1518,E2 108.0966} C_DIS
LIN {X 86.3563,Y -32.4294,Z 94,A -25.8429,B 24.9264,C -1.9815,E1 25.1491,E2 111.0076} C_DIS
LIN {X 84.506,Y -36.9837,Z 94,A -28.8194,B 24.9269,C -1.975,E1 25.1459,E2 113.983} C_DIS
LIN {X 82.7704,Y -40.7207,Z 94,A -31.5794,B 24.928,C -1.96,E1 25.1425,E2 116.7636} C_DIS
LIN {X 80.9545,Y -44.2208,Z 94,A -33.7691,B 24.9278,C -1.9623,E1 25.1397,E2 118.9363} C_DIS
LIN {X 79.3805,Y -46.9869,Z 94,A -36.0712,B 24.9291,C -1.9447,E1 25.1364,E2 121.2681} C_DIS
LIN {X 76.8576,Y -51.0099,Z 94,A -38.6456,B 24.9287,C -1.95,E1 25.1326,E2 123.8169} C_DIS
LIN {X 74.9656,Y -53.7516,Z 94,A -40.8053,B 24.9294,C -1.941,E1 25.1291,E2 125.9874} C_DIS
LIN {X 72.0153,Y -57.6454,Z 94,A -44.4566,B 24.9316,C -1.9106,E1 25.1227,E2 129.6933} C_DIS
LIN {X 69.4443,Y -60.7167,Z 94,A -46.1158,B 24.9299,C -1.9341,E1 25.1198,E2 131.2894} C_DIS
LIN {X 67.4197,Y -62.9581,Z 94,A -48.7703,B 24.9322,C -1.9013,E1 25.1146,E2 134.0097} C_DIS
LIN {X 64.6717,Y -65.7773,Z 94,A -50.5226,B 24.9309,C -1.9203,E1 25.1113,E2 135.7098} C_DIS
LIN {X 61.9722,Y -68.3284,Z 94,A -52.8835,B 24.9314,C -1.9129,E1 25.1064,E2 138.0785} C_DIS
LIN {X 59.426,Y -70.5539,Z 94,A -55.5021,B 24.9331,C -1.8897,E1 25.1008,E2 140.742} C_DIS
LIN {X 56.6132,Y -72.8295,Z 94,A -57.3793,B 24.9325,C -1.898,E1 25.0967,E2 142.5925} C_DIS
LIN {X 53.8372,Y -74.9045,Z 94,A -59.3253,B 24.9323,C -1.9009,E1 25.0923,E2 144.5247} C_DIS
LIN {X 50.9808,Y -76.8768,Z 94,A -61.4747,B 24.9325,C -1.8969,E1 25.0873,E2 146.6764} C_DIS
LIN {X 47.3039,Y -79.1932,Z 94,A -64.1414,B 24.9328,C -1.8929,E1 25.081,E2 149.344} C_DIS
LIN {X 45.3159,Y -80.3471,Z 94,A -65.5705,B 24.933,C -1.8903,E1 25.0775,E2 150.775} C_DIS
LIN {X 41.5819,Y -82.3411,Z 94,A -68.3566,B 24.9337,C -1.8803,E1 25.0706,E2 153.577} C_DIS
LIN {X 36.4606,Y -84.7339,Z 94,A -71.6128,B 24.9335,C -1.8839,E1 25.0624,E2 156.8166} C_DIS
LIN {X 33.5447,Y -85.9292,Z 94,A -73.7506,B 24.9341,C -1.8748,E1 25.0568,E2 158.971} C_DIS
LIN {X 30.6396,Y -87.0072,Z 94,A -75.4431,B 24.9337,C -1.8805,E1 25.0524,E2 160.6467} C_DIS
LIN {X 27.9016,Y -87.925,Z 94,A -77.4323,B 24.9343,C -1.8714,E1 25.0471,E2 162.6535} C_DIS
LIN {X 23.7307,Y -89.1404,Z 94,A -80.2397,B 24.9348,C -1.8647,E1 25.0395,E2 165.4722} C_DIS
LIN {X 18.2824,Y -90.4149,Z 94,A -83.5093,B 24.9345,C -1.8686,E1 25.0306,E2 168.7281} C_DIS
LIN {X 10.8235,Y -91.6073,Z 94,A -89.3793,B 24.9375,C -1.8255,E1 25.0141,E2 174.6953} C_DIS
LIN {X 5.0684,Y -92.1051,Z 94,A -91.2898,B 24.9337,C -1.8807,E1 25.0092,E2 176.474} C_DIS
LIN {X 0.6403,Y -92.241,Z 94,A -94.4247,B 24.9347,C -1.8667,E1 25.0003,E2 179.6414} C_DIS
Enddeposition()
LIN {X 0.6403,Y -92.241,Z 94,A -94.4247,B 24.9347,C -1.8667,E1 25.0003,E2 179.6414} C_DIS
Startdeposition()
$VEL.CP = VEL_PRINT
LIN {X 3.8275,Y -91.23,Z 94,A -91.5975,B 24.9315,C -1.9118,E1 25.0085,E2 176.7079} C_DIS
LIN {X 7.8808,Y -90.971,Z 94,A -88.6137,B 24.9303,C -1.928,E1 25.0169,E2 173.6872} C_DIS
LIN {X 12.7075,Y -90.4218,Z 94,A -85.6804,B 24.9305,C -1.9259,E1 25.025,E2 170.7611} C_DIS
LIN {X 17.28,Y -89.6603,Z 94,A -83.1851,B 24.9313,C -1.9139,E1 25.0318,E2 168.2971} C_DIS
LIN {X 20.3732,Y -89.0086,Z 94,A -81.2636,B 24.9313,C -1.9135,E1 25.037,E2 166.3789} C_DIS
LIN {X 24.5708,Y -87.9428,Z 94,A -78.3707,B 24.9307,C -1.9225,E1 25.0449,E2 163.4694} C_DIS
LIN {X 27.4616,Y -87.084,Z 94,A -76.4479,B 24.9305,C -1.9257,E1 25.05,E2 161.5424} C_DIS
LIN {X 30.7188,Y -85.9893,Z 94,A -74.4079,B 24.9305,C -1.9244,E1 25.0554,E2 159.5096} C_DIS
LIN {X 34.9641,Y -84.3526,Z 94,A -71.7026,B 24.9307,C -1.923,E1 25.0624,E2 156.8135} C_DIS
LIN {X 39.2845,Y -82.428,Z 94,A -68.0288,B 24.9285,C -1.9528,E1 25.0719,E2 153.0786} C_DIS
LIN {X 42.4414,Y -80.8474,Z 94,A -66.3855,B 24.9297,C -1.936,E1 25.0758,E2 151.4795} C_DIS
LIN {X 45.4092,Y -79.2186,Z 94,A -64.2773,B 24.9295,C -1.9392,E1 25.0809,E2 149.37} C_DIS
LIN {X 48.1116,Y -77.6075,Z 94,A -62.2724,B 24.9291,C -1.944,E1 25.0857,E2 147.3601} C_DIS
LIN {X 50.9594,Y -75.7679,Z 94,A -60.2016,B 24.929,C -1.9461,E1 25.0906,E2 145.291} C_DIS
LIN {X 53.737,Y -73.8239,Z 94,A -58.0745,B 24.9287,C -1.9505,E1 25.0954,E2 143.161} C_DIS
LIN {X 55.6272,Y -72.4099,Z 94,A -56.6967,B 24.9287,C -1.9499,E1 25.0985,E2 141.7896} C_DIS
LIN {X 58.1182,Y -70.4268,Z 94,A -54.6198,B 24.9282,C -1.9572,E1 25.103,E2 139.7035} C_DIS
LIN {X 60.5805,Y -68.3209,Z 94,A -52.5416,B 24.9277,C -1.9634,E1 25.1074,E2 137.6186} C_DIS
LIN {X 62.9657,Y -66.1301,Z 94,A -50.6997,B 24.9279,C -1.9613,E1 25.1111,E2 135.7893} C_DIS
LIN {X 64.8658,Y -64.2651,Z 94,A -48.7439,B 24.9268,C -1.9758,E1 25.115,E2 133.8076} C_DIS
LIN {X 67.5009,Y -61.4922,Z 94,A -46.4523,B 24.9267,C -1.9778,E1 25.1194,E2 131.5213} C_DIS
LIN {X 69.5982,Y -59.1073,Z 94,A -44.6277,B 24.9267,C -1.9768,E1 25.1227,E2 129.7073} C_DIS
LIN {X 71.7999,Y -56.4128,Z 94,A -42.2888,B 24.9259,C -1.9883,E1 25.1268,E2 127.3522} C_DIS
LIN {X 73.9279,Y -53.5949,Z 94,A -40.0926,B 24.9255,C -1.9935,E1 25.1304,E2 125.1541} C_DIS
LIN {X 75.8732,Y -50.8039,Z 94,A -37.981,B 24.9251,C -1.9986,E1 25.1338,E2 123.0409} C_DIS
LIN {X 77.6536,Y -48.0378,Z 94,A -35.9063,B 24.9246,C -2.0049,E1 25.1369,E2 120.9619} C_DIS
LIN {X 79.4084,Y -45.0787,Z 94,A -33.972,B 24.9248,C -2.0029,E1 25.1396,E2 119.0424} C_DIS
LIN {X 80.8846,Y -42.3708,Z 94,A -32.1714,B 24.9248,C -2.0036,E1 25.1419,E2 117.2495} C_DIS
LIN {X 82.7996,Y -38.494,Z 94,A -29.3668,B 24.9239,C -2.015,E1 25.1454,E2 114.433} C_DIS
LIN {X 84.7305,Y -34.0364,Z 94,A -25.6895,B 24.9214,C -2.0476,E1 25.1494,E2 110.699} C_DIS
LIN {X 85.9109,Y -30.9354,Z 94,A -24.1025,B 24.9223,C -2.0356,E1 25.1509,E2 109.1491} C_DIS
LIN {X 86.9547,Y -27.8659,Z 94,A -22.0236,B 24.9217,C -2.0436,E1 25.1527,E2 107.063} C_DIS
LIN {X 88.0197,Y -24.2969,Z 94,A -19.533,B 24.9207,C -2.0567,E1 25.1546,E2 104.5559} C_DIS
LIN {X 89.0919,Y -20.0123,Z 94,A -16.9346,B 24.9205,C -2.059,E1 25.1563,E2 101.9671} C_DIS
LIN {X 90.1624,Y -14.4411,Z 94,A -13.4674,B 24.9199,C -2.067,E1 25.158,E2 98.5014} C_DIS
LIN {X 90.896,Y -8.693,Z 94,A -9.8677,B 24.9191,C -2.0773,E1 25.1592,E2 94.8987} C_DIS
LIN {X 91.1553,Y -5.3253,Z 94,A -7.8139,B 24.9187,C -2.0817,E1 25.1596,E2 92.8467} C_DIS
LIN {X 91.2649,Y -2.8797,Z 94,A -5.2761,B 24.9154,C -2.124,E1 25.1598,E2 90.2241} C_DIS
LIN {X 91.2863,Y 2.1398,Z 94,A -3.3018,B 24.9181,C -2.0902,E1 25.1598,E2 88.3412} C_DIS
LIN {X 91.1149,Y 5.9723,Z 94,A -0.4453,B 24.9161,C -2.1146,E1 25.1593,E2 85.4442} C_DIS
LIN {X 90.8086,Y 9.558,Z 94,A 2.0506,B 24.9149,C -2.1306,E1 25.1586,E2 82.9254} C_DIS
LIN {X 90.379,Y 13.0089,Z 94,A 3.6539,B 24.916,C -2.116,E1 25.158,E2 81.366} C_DIS
LIN {X 89.8888,Y 16.0492,Z 94,A 5.6703,B 24.9153,C -2.1251,E1 25.157,E2 79.3398} C_DIS
LIN {X 89.3625,Y 18.7636,Z 94,A 7.4673,B 24.9147,C -2.1328,E1 25.156,E2 77.5353} C_DIS
LIN {X 88.5357,Y 22.3416,Z 94,A 9.683,B 24.9144,C -2.1366,E1 25.1545,E2 75.3234} C_DIS
LIN {X 87.7272,Y 25.3319,Z 94,A 11.6072,B 24.914,C -2.1417,E1 25.1531,E2 73.398} C_DIS
LIN {X 86.7263,Y 28.5718,Z 94,A 13.9195,B 24.9129,C -2.1549,E1 25.1511,E2 71.0678} C_DIS
LIN {X 85.2986,Y 32.585,Z 94,A 16.3392,B 24.913,C -2.1534,E1 25.1488,E2 68.665} C_DIS
LIN {X 84.4605,Y 34.6998,Z 94,A 17.9911,B 24.912,C -2.1658,E1 25.147,E2 66.993} C_DIS
LIN {X 82.71,Y 38.6864,Z 94,A 20.5162,B 24.912,C -2.166,E1 25.1441,E2 64.4813} C_DIS
LIN {X 81.3148,Y 41.5387,Z 94,A 22.3516,B 24.912,C -2.1658,E1 25.1418,E2 62.6561} C_DIS
LIN {X 78.702,Y 46.299,Z 94,A 25.8136,B 24.9111,C -2.1769,E1 25.1371,E2 59.1858} C_DIS
LIN {X 77.1592,Y 48.8294,Z 94,A 27.7861,B 24.9104,C -2.1858,E1 25.1341,E2 57.2021} C_DIS
LIN {X 75.6,Y 51.2074,Z 94,A 29.617,B 24.9099,C -2.1921,E1 25.1313,E2 55.3656} C_DIS
LIN {X 72.3578,Y 55.6948,Z 94,A 33.3116,B 24.9085,C -2.2086,E1 25.1251,E2 51.6497} C_DIS
LIN {X 69.4106,Y 59.3274,Z 94,A 35.7321,B 24.9095,C -2.1969,E1 25.1208,E2 49.268} C_DIS
LIN {X 66.985,Y 62.0545,Z 94,A 38.1669,B 24.9086,C -2.2072,E1 25.1162,E2 46.8196} C_DIS
LIN {X 64.6959,Y 64.4372,Z 94,A 40.1931,B 24.9084,C -2.21,E1 25.1123,E2 44.7955} C_DIS
LIN {X 62.2221,Y 66.8294,Z 94,A 42.3841,B 24.9079,C -2.2155,E1 25.1078,E2 42.6003} C_DIS
LIN {X 59.9549,Y 68.8694,Z 94,A 44.3051,B 24.9076,C -2.2196,E1 25.1038,E2 40.6774} C_DIS
LIN {X 57.4194,Y 70.997,Z 94,A 46.331,B 24.9074,C -2.2217,E1 25.0994,E2 38.6543} C_DIS
LIN {X 55.3493,Y 72.6241,Z 94,A 48.4398,B 24.9058,C -2.2408,E1 25.0947,E2 36.5079} C_DIS
LIN {X 52.6176,Y 74.6272,Z 94,A 50.0704,B 24.907,C -2.2269,E1 25.091,E2 34.9159} C_DIS
LIN {X 50.3331,Y 76.185,Z 94,A 52.988,B 24.9032,C -2.2715,E1 25.084,E2 31.9022} C_DIS
LIN {X 45.3912,Y 79.2289,Z 94,A 55.3344,B 24.9066,C -2.2311,E1 25.0786,E2 29.6588} C_DIS
LIN {X 42.4819,Y 80.8261,Z 94,A 57.6336,B 24.9058,C -2.2414,E1 25.0729,E2 27.3417} C_DIS
LIN {X 38.9386,Y 82.5927,Z 94,A 60.041,B 24.9058,C -2.2418,E1 25.0669,E2 24.9398} C_DIS
LIN {X 35.8296,Y 83.9879,Z 94,A 62.0716,B 24.9058,C -2.2404,E1 25.0617,E2 22.9173} C_DIS
LIN {X 33.3941,Y 84.9847,Z 94,A 64.3283,B 24.9039,C -2.263,E1 25.0557,E2 20.6121} C_DIS
LIN {X 29.9614,Y 86.2552,Z 94,A 66.1034,B 24.9053,C -2.247,E1 25.0511,E2 18.8785} C_DIS
LIN {X 26.2826,Y 87.4465,Z 94,A 68.4089,B 24.9055,C -2.2447,E1 25.045,E2 16.5826} C_DIS
LIN {X 23.4036,Y 88.261,Z 94,A 70.4254,B 24.905,C -2.2507,E1 25.0395,E2 14.5552} C_DIS
LIN {X 19.8399,Y 89.1296,Z 94,A 72.6474,B 24.905,C -2.2492,E1 25.0335,E2 12.3398} C_DIS
LIN {X 17.0306,Y 89.7083,Z 94,A 74.4499,B 24.905,C -2.2501,E1 25.0286,E2 10.5374} C_DIS
LIN {X 14.2849,Y 90.1866,Z 94,A 76.1682,B 24.905,C -2.2496,E1 25.0239,E2 8.8219} C_DIS
LIN {X 11.0893,Y 90.6356,Z 94,A 78.0048,B 24.9056,C -2.2438,E1 25.0188,E2 7.0008} C_DIS
LIN {X 8.3794,Y 90.9249,Z 94,A 79.9251,B 24.9049,C -2.251,E1 25.0134,E2 5.0644} C_DIS
LIN {X 5.6876,Y 91.1342,Z 94,A 81.7774,B 24.9045,C -2.2563,E1 25.0082,E2 3.2004} C_DIS
LIN {X 1.7066,Y 91.2943,Z 94,A 84.0816,B 24.9051,C -2.2496,E1 25.0019,E2 0.9127} C_DIS
LIN {X -1.9669,Y 91.2895,Z 94,A 86.8347,B 24.9039,C -2.2639,E1 24.9941,E2 -1.8745} C_DIS
LIN {X -6.8793,Y 91.0516,Z 94,A 89.5173,B 24.9051,C -2.2493,E1 24.9867,E2 -4.5234} C_DIS
LIN {X -10.1914,Y 90.7408,Z 94,A 91.6798,B 24.905,C -2.2507,E1 24.9807,E2 -6.6904} C_DIS
LIN {X -14.3605,Y 90.1749,Z 94,A 94.2448,B 24.9053,C -2.2465,E1 24.9736,E2 -9.2476} C_DIS
LIN {X -18.0597,Y 89.507,Z 94,A 96.6455,B 24.9053,C -2.246,E1 24.967,E2 -11.6497} C_DIS
LIN {X -21.6561,Y 88.705,Z 94,A 98.8408,B 24.9059,C -2.2401,E1 24.9611,E2 -13.8339} C_DIS
LIN {X -24.7873,Y 87.8815,Z 94,A 100.6277,B 24.9067,C -2.2302,E1 24.9563,E2 -15.5999} C_DIS
LIN {X -27.7105,Y 87.005,Z 94,A 102.9144,B 24.9059,C -2.2399,E1 24.9501,E2 -17.9136} C_DIS
LIN {X -30.638,Y 86.0178,Z 94,A 105.0598,B 24.9055,C -2.2441,E1 24.9444,E2 -20.0733} C_DIS
LIN {X -34.3408,Y 84.6066,Z 94,A 107.2284,B 24.9067,C -2.2306,E1 24.9389,E2 -22.2145} C_DIS
LIN {X -37.2019,Y 83.3888,Z 94,A 109.2708,B 24.9067,C -2.2306,E1 24.9336,E2 -24.2618} C_DIS
LIN {X -39.8428,Y 82.1597,Z 94,A 111.05,B 24.907,C -2.2263,E1 24.9292,E2 -26.035} C_DIS
LIN {X -42.5828,Y 80.773,Z 94,A 112.8341,B 24.9077,C -2.2186,E1 24.9248,E2 -27.8058} C_DIS
LIN {X -46.0826,Y 78.8299,Z 94,A 115.6518,B 24.9072,C -2.2238,E1 24.9179,E2 -30.6441} C_DIS
LIN {X -49.609,Y 76.6591,Z 94,A 118.2644,B 24.9076,C -2.2194,E1 24.9117,E2 -33.2545} C_DIS
LIN {X -52.5595,Y 74.6682,Z 94,A 120.53,B 24.9079,C -2.216,E1 24.9065,E2 -35.5196} C_DIS
LIN {X -55.5506,Y 72.4689,Z 94,A 122.5028,B 24.9092,C -2.2,E1 24.9022,E2 -37.4615} C_DIS
LIN {X -58.0411,Y 70.4909,Z 94,A 124.7503,B 24.9089,C -2.2035,E1 24.8972,E2 -39.7257} C_DIS
LIN {X -60.4883,Y 68.4035,Z 94,A 126.8941,B 24.9089,C -2.2028,E1 24.8927,E2 -41.8763} C_DIS
LIN {X -63.1898,Y 65.9141,Z 94,A 129.1345,B 24.9096,C -2.1955,E1 24.8882,E2 -44.1083} C_DIS
LIN {X -65.792,Y 63.3165,Z 94,A 131.4723,B 24.91,C -2.1908,E1 24.8836,E2 -46.445} C_DIS
LIN {X -67.9979,Y 60.9414,Z 94,A 133.4112,B 24.9106,C -2.1828,E1 24.88,E2 -48.3735} C_DIS
LIN {X -70.1157,Y 58.4926,Z 94,A 135.5119,B 24.9109,C -2.1797,E1 24.8762,E2 -50.4764} C_DIS
LIN {X -72.3668,Y 55.6831,Z 94,A 137.8323,B 24.9112,C -2.1756,E1 24.8722,E2 -52.798} C_DIS
LIN {X -74.4546,Y 52.8595,Z 94,A 140.0835,B 24.9116,C -2.1711,E1 24.8685,E2 -55.0494} C_DIS
LIN {X -76.1699,Y 50.356,Z 94,A 142.4775,B 24.9108,C -2.1808,E1 24.8647,E2 -57.4785} C_DIS
LIN {X -78.0658,Y 47.3634,Z 94,A 143.9193,B 24.9132,C -2.1507,E1 24.8627,E2 -58.8558} C_DIS
LIN {X -80.5505,Y 43.0051,Z 94,A 147.6856,B 24.9125,C -2.1603,E1 24.8576,E2 -62.6647} C_DIS
LIN {X -82.7264,Y 38.6512,Z 94,A 150.3593,B 24.9141,C -2.1397,E1 24.8543,E2 -65.3038} C_DIS
LIN {X -84.0539,Y 35.6729,Z 94,A 152.4645,B 24.9145,C -2.1353,E1 24.852,E2 -67.4101} C_DIS
LIN {X -85.3022,Y 32.5754,Z 94,A 154.5791,B 24.915,C -2.1295,E1 24.8498,E2 -69.5226} C_DIS
LIN {X -86.4683,Y 29.3397,Z 94,A 156.8807,B 24.9151,C -2.1271,E1 24.8477,E2 -71.8318} C_DIS
LIN {X -87.4708,Y 26.2007,Z 94,A 158.8456,B 24.9159,C -2.1176,E1 24.8461,E2 -73.7851} C_DIS
LIN {X -88.4272,Y 22.7639,Z 94,A 161.0299,B 24.9166,C -2.1089,E1 24.8445,E2 -75.9615} C_DIS
LIN {X -89.116,Y 19.9023,Z 94,A 162.9616,B 24.9169,C -2.1056,E1 24.8433,E2 -77.8966} C_DIS
LIN {X -89.6241,Y 17.4681,Z 94,A 164.4521,B 24.9174,C -2.0985,E1 24.8425,E2 -79.379} C_DIS
LIN {X -90.1452,Y 14.5488,Z 94,A 166.3991,B 24.9177,C -2.0952,E1 24.8416,E2 -81.3296} C_DIS
LIN {X -90.5806,Y 11.5226,Z 94,A 168.3463,B 24.9181,C -2.0899,E1 24.8409,E2 -83.2759} C_DIS
LIN {X -90.9379,Y 8.239,Z 94,A 170.4258,B 24.9186,C -2.0835,E1 24.8403,E2 -85.3525} C_DIS
LIN {X -91.1992,Y 4.5305,Z 94,A 172.8652,B 24.9189,C -2.0792,E1 24.8399,E2 -87.7963} C_DIS
LIN {X -91.305,Y 1.1206,Z 94,A 175.0237,B 24.9194,C -2.0728,E1 24.8398,E2 -89.9526} C_DIS
LIN {X -91.2863,Y -2.1393,Z 94,A 176.9079,B 24.9203,C -2.0614,E1 24.8398,E2 -91.821} C_DIS
LIN {X -91.201,Y -4.4976,Z 94,A 178.6711,B 24.92,C -2.0652,E1 24.8401,E2 -93.6039} C_DIS
LIN {X -90.97,Y -7.8912,Z 94,A -179.3472,B 24.9209,C -2.0538,E1 24.8405,E2 -95.5703} C_DIS
LIN {X -90.6143,Y -11.2625,Z 94,A -177.1619,B 24.9213,C -2.0489,E1 24.8412,E2 -97.7568} C_DIS
LIN {X -90.1609,Y -14.4509,Z 94,A -175.0845,B 24.9216,C -2.0443,E1 24.8421,E2 -99.8356} C_DIS
LIN {X -89.6338,Y -17.4172,Z 94,A -173.2577,B 24.9222,C -2.0365,E1 24.8431,E2 -101.6546} C_DIS
LIN {X -88.9546,Y -20.6068,Z 94,A -171.2833,B 24.9229,C -2.028,E1 24.8443,E2 -103.6204} C_DIS
LIN {X -88.1387,Y -23.8565,Z 94,A -169.2188,B 24.9235,C -2.0204,E1 24.8457,E2 -105.6789} C_DIS
LIN {X -87.2474,Y -26.9346,Z 94,A -167.1553,B 24.9238,C -2.016,E1 24.8474,E2 -107.7437} C_DIS
LIN {X -86.6005,Y -28.9478,Z 94,A -165.657,B 24.9237,C -2.0173,E1 24.8487,E2 -109.2535} C_DIS
LIN {X -85.4589,Y -32.1617,Z 94,A -163.5844,B 24.9243,C -2.0089,E1 24.8507,E2 -111.318} C_DIS
LIN {X -83.797,Y -36.2722,Z 94,A -160.7977,B 24.9249,C -2.0011,E1 24.8537,E2 -114.1014} C_DIS
LIN {X -82.3259,Y -39.497,Z 94,A -158.5926,B 24.9254,C -1.9942,E1 24.8563,E2 -116.3022} C_DIS
LIN {X -80.6504,Y -42.8154,Z 94,A -156.1788,B 24.9257,C -1.9903,E1 24.8594,E2 -118.7195} C_DIS
LIN {X -78.9765,Y -45.8304,Z 94,A -154.2649,B 24.9267,C -1.9768,E1 24.862,E2 -120.6113} C_DIS
LIN {X -77.3087,Y -48.5901,Z 94,A -152.1375,B 24.9269,C -1.9747,E1 24.8651,E2 -122.7446} C_DIS
LIN {X -75.7771,Y -50.9459,Z 94,A -150.1859,B 24.9268,C -1.976,E1 24.8681,E2 -124.7091} C_DIS
LIN {X -73.4921,Y -54.1901,Z 94,A -148.0064,B 24.928,C -1.9602,E1 24.8716,E2 -126.8616} C_DIS
LIN {X -71.3951,Y -56.925,Z 94,A -145.5883,B 24.9278,C -1.963,E1 24.8758,E2 -129.2977} C_DIS
LIN {X -69.4634,Y -59.2655,Z 94,A -143.6568,B 24.928,C -1.9595,E1 24.8792,E2 -131.2297} C_DIS
LIN {X -67.3027,Y -61.7083,Z 94,A -141.6068,B 24.9283,C -1.955,E1 24.8831,E2 -133.2782} C_DIS
LIN {X -65.0365,Y -64.0923,Z 94,A -139.5356,B 24.9287,C -1.9508,E1 24.8871,E2 -135.3482} C_DIS
LIN {X -62.445,Y -66.6198,Z 94,A -137.1768,B 24.9287,C -1.9489,E1 24.8919,E2 -137.7123} C_DIS
LIN {X -59.6338,Y -69.1496,Z 94,A -134.4274,B 24.9283,C -1.9562,E1 24.8977,E2 -140.49} C_DIS
LIN {X -55.8761,Y -72.2181,Z 94,A -131.7842,B 24.9296,C -1.9379,E1 24.9034,E2 -143.0994} C_DIS
LIN {X -53.3545,Y -74.1014,Z 94,A -129.781,B 24.9298,C -1.9354,E1 24.9079,E2 -145.1037} C_DIS
LIN {X -50.9154,Y -75.7977,Z 94,A -127.4298,B 24.9288,C -1.9481,E1 24.9135,E2 -147.4929} C_DIS
LIN {X -48.0232,Y -77.6628,Z 94,A -125.8421,B 24.9304,C -1.9264,E1 24.9171,E2 -149.0339} C_DIS
LIN {X -45.4758,Y -79.1803,Z 94,A -123.8268,B 24.9303,C -1.9287,E1 24.922,E2 -151.0609} C_DIS
LIN {X -42.0768,Y -81.0394,Z 94,A -121.3992,B 24.9305,C -1.9254,E1 24.928,E2 -153.4873} C_DIS
LIN {X -38.8883,Y -82.6161,Z 94,A -119.4898,B 24.9314,C -1.9123,E1 24.9327,E2 -155.3705} C_DIS
LIN {X -36.5125,Y -83.6923,Z 94,A -117.0117,B 24.9296,C -1.9381,E1 24.9392,E2 -157.9158} C_DIS
LIN {X -33.1066,Y -85.0976,Z 94,A -115.2223,B 24.931,C -1.9186,E1 24.9438,E2 -159.6628} C_DIS
LIN {X -29.5725,Y -86.3898,Z 94,A -112.8168,B 24.931,C -1.9181,E1 24.9501,E2 -162.0718} C_DIS
LIN {X -26.5782,Y -87.3579,Z 94,A -111.0891,B 24.9317,C -1.9084,E1 24.9546,E2 -163.7796} C_DIS
LIN {X -23.9382,Y -88.1166,Z 94,A -109.2463,B 24.9315,C -1.9113,E1 24.9596,E2 -165.6321} C_DIS
LIN {X -21.1056,Y -88.8392,Z 94,A -107.2418,B 24.9312,C -1.916,E1 24.9651,E2 -167.6504} C_DIS
LIN {X -17.7209,Y -89.5754,Z 94,A -105.1551,B 24.9315,C -1.9121,E1 24.9708,E2 -169.7305} C_DIS
LIN {X -14.2462,Y -90.1925,Z 94,A -103.0955,B 24.9319,C -1.9063,E1 24.9764,E2 -171.7782} C_DIS
LIN {X -11.2267,Y -90.6189,Z 94,A -101.0304,B 24.9315,C -1.911,E1 24.9822,E2 -173.8559} C_DIS
LIN {X -8.8412,Y -90.8823,Z 94,A -99.1122,B 24.9305,C -1.9248,E1 24.9876,E2 -175.8081} C_DIS
LIN {X -5.6321,Y -91.1379,Z 94,A -97.5852,B 24.9317,C -1.9081,E1 24.9918,E2 -177.2959} C_DIS
LIN {X -0.9531,Y -91.3061,Z 94,A -94.5599,B 24.9315,C -1.9115,E1 25.0002,E2 -180.3296} C_DIS
LIN {X -0.9531,Y -91.3061,Z 94,A -94.5599,B 24.9315,C -1.9115,E1 25.0002,E2 -180.3296} C_DIS
Enddeposition()
LIN {X 0.6412,Y -90.373,Z 94,A -94.514,B 24.9326,C -1.8959,E1 25.0002,E2 -180.3385} C_DIS
Startdeposition()
$VEL.CP = VEL_PRINT
LIN {X -2.5208,Y -90.3413,Z 94,A -96.6007,B 24.9328,C -1.8928,E1 24.9944,E2 -178.2444} C_DIS
LIN {X -5.2705,Y -90.2227,Z 94,A -98.2132,B 24.9325,C -1.8971,E1 24.9899,E2 -176.6416} C_DIS
LIN {X -7.4988,Y -90.0649,Z 94,A -99.6408,B 24.9325,C -1.8967,E1 24.986,E2 -175.2125} C_DIS
LIN {X -10.7933,Y -89.7297,Z 94,A -101.7452,B 24.9325,C -1.8968,E1 24.9801,E2 -173.1071} C_DIS
LIN {X -14.0941,Y -89.2708,Z 94,A -103.8527,B 24.9325,C -1.8975,E1 24.9743,E2 -170.9993} C_DIS
LIN {X -16.2746,Y -88.8991,Z 94,A -105.2544,B 24.9325,C -1.898,E1 24.9704,E2 -169.5975} C_DIS
LIN {X -19.5268,Y -88.2418,Z 94,A -107.3688,B 24.9325,C -1.8985,E1 24.9646,E2 -167.4819} C_DIS
LIN {X -22.2353,Y -87.5985,Z 94,A -109.2346,B 24.9325,C -1.8962,E1 24.9596,E2 -165.6079} C_DIS
LIN {X -24.9106,Y -86.8756,Z 94,A -110.8868,B 24.9323,C -1.9007,E1 24.9551,E2 -163.9639} C_DIS
LIN {X -27.2933,Y -86.1581,Z 94,A -112.4349,B 24.9321,C -1.9028,E1 24.951,E2 -162.418} C_DIS
LIN {X -29.1352,Y -85.5514,Z 94,A -113.6993,B 24.9321,C -1.9027,E1 24.9477,E2 -161.1509} C_DIS
LIN {X -32.0648,Y -84.4966,Z 94,A -115.7554,B 24.9321,C -1.9018,E1 24.9423,E2 -159.0886} C_DIS
LIN {X -35.0302,Y -83.311,Z 94,A -117.7625,B 24.9321,C -1.9044,E1 24.9371,E2 -157.0831} C_DIS
LIN {X -37.6451,Y -82.1643,Z 94,A -119.4866,B 24.9317,C -1.9091,E1 24.9327,E2 -155.366} C_DIS
LIN {X -39.6447,Y -81.2184,Z 94,A -120.8918,B 24.9316,C -1.9106,E1 24.9292,E2 -153.9609} C_DIS
LIN {X -42.5995,Y -79.7083,Z 94,A -123.2253,B 24.9319,C -1.9061,E1 24.9233,E2 -151.6103} C_DIS
LIN {X -45.5109,Y -78.0826,Z 94,A -125.345,B 24.9317,C -1.9089,E1 24.9182,E2 -149.4908} C_DIS
LIN {X -48.3796,Y -76.3382,Z 94,A -127.2567,B 24.931,C -1.9188,E1 24.9137,E2 -147.5969} C_DIS
LIN {X -50.7154,Y -74.805,Z 94,A -129.1349,B 24.931,C -1.9183,E1 24.9093,E2 -145.7113} C_DIS
LIN {X -52.9472,Y -73.2443,Z 94,A -130.7677,B 24.9306,C -1.9241,E1 24.9056,E2 -144.0866} C_DIS
LIN {X -55.1591,Y -71.5912,Z 94,A -132.6374,B 24.9306,C -1.9235,E1 24.9014,E2 -142.2087} C_DIS
LIN {X -57.7464,Y -69.5211,Z 94,A -134.7489,B 24.9304,C -1.9271,E1 24.8969,E2 -140.0977} C_DIS
LIN {X -60.2885,Y -67.3285,Z 94,A -136.8858,B 24.9301,C -1.9309,E1 24.8924,E2 -137.9617} C_DIS
LIN {X -62.7221,Y -65.0674,Z 94,A -138.9993,B 24.9298,C -1.935,E1 24.8881,E2 -135.8491} C_DIS
LIN {X -65.0713,Y -62.7181,Z 94,A -141.1156,B 24.9295,C -1.9392,E1 24.8839,E2 -133.7338} C_DIS
LIN {X -67.3325,Y -60.2841,Z 94,A -143.2333,B 24.9292,C -1.9435,E1 24.88,E2 -131.617} C_DIS
LIN {X -69.5025,Y -57.7688,Z 94,A -145.3514,B 24.9289,C -1.948,E1 24.8761,E2 -129.4998} C_DIS
LIN {X -71.6,Y -55.1478,Z 94,A -147.443,B 24.9284,C -1.9541,E1 24.8725,E2 -127.4131} C_DIS
LIN {X -73.2544,Y -52.9332,Z 94,A -149.1348,B 24.928,C -1.9602,E1 24.8697,E2 -125.7277} C_DIS
LIN {X -74.9922,Y -50.4389,Z 94,A -151.0792,B 24.9276,C -1.9646,E1 24.8667,E2 -123.784} C_DIS
LIN {X -76.2027,Y -48.5906,Z 94,A -152.4881,B 24.9274,C -1.9679,E1 24.8645,E2 -122.376} C_DIS
LIN {X -77.3675,Y -46.7137,Z 94,A -153.9336,B 24.9272,C -1.9702,E1 24.8624,E2 -120.9286} C_DIS
LIN {X -79.0418,Y -43.8213,Z 94,A -156.2526,B 24.9272,C -1.9699,E1 24.8592,E2 -118.5968} C_DIS
LIN {X -80.6854,Y -40.7175,Z 94,A -158.277,B 24.9263,C -1.982,E1 24.8566,E2 -116.5904} C_DIS
LIN {X -82.0533,Y -37.8835,Z 94,A -160.2758,B 24.9259,C -1.9875,E1 24.8542,E2 -114.5938} C_DIS
LIN {X -83.0661,Y -35.6112,Z 94,A -161.8724,B 24.9256,C -1.9914,E1 24.8524,E2 -112.9977} C_DIS
LIN {X -83.9196,Y -33.5505,Z 94,A -163.2814,B 24.9253,C -1.9956,E1 24.8509,E2 -111.591} C_DIS
LIN {X -84.7132,Y -31.493,Z 94,A -164.6931,B 24.9251,C -1.9993,E1 24.8495,E2 -110.1801} C_DIS
LIN {X -85.6917,Y -28.7193,Z 94,A -166.7768,B 24.9251,C -1.9984,E1 24.8476,E2 -108.0823} C_DIS
LIN {X -86.7248,Y -25.4309,Z 94,A -168.8035,B 24.9243,C -2.0096,E1 24.846,E2 -106.0708} C_DIS
LIN {X -87.3935,Y -23.033,Z 94,A -170.3583,B 24.9239,C -2.0151,E1 24.8449,E2 -104.5199} C_DIS
LIN {X -88.119,Y -20.0735,Z 94,A -172.4985,B 24.9239,C -2.0149,E1 24.8435,E2 -102.3667} C_DIS
LIN {X -88.7983,Y -16.8157,Z 94,A -174.4645,B 24.9231,C -2.0256,E1 24.8424,E2 -100.4148} C_DIS
LIN {X -89.1853,Y -14.6252,Z 94,A -175.8809,B 24.9227,C -2.0299,E1 24.8417,E2 -99.0001} C_DIS
LIN {X -89.5554,Y -12.1643,Z 94,A -177.4372,B 24.9223,C -2.0354,E1 24.8411,E2 -97.4478} C_DIS
LIN {X -89.8265,Y -9.967,Z 94,A -178.8508,B 24.922,C -2.0396,E1 24.8407,E2 -96.0356} C_DIS
LIN {X -90.0184,Y -8.0374,Z 94,A 179.8768,B 24.9218,C -2.0422,E1 24.8403,E2 -94.7619} C_DIS
LIN {X -90.2236,Y -5.2544,Z 94,A 177.9861,B 24.9216,C -2.0443,E1 24.84,E2 -92.8647} C_DIS
LIN {X -90.3422,Y -2.489,Z 94,A 176.3306,B 24.921,C -2.0528,E1 24.8398,E2 -91.2196} C_DIS
LIN {X -90.3742,Y 0.6546,Z 94,A 174.2814,B 24.9206,C -2.0575,E1 24.8398,E2 -89.1693} C_DIS
LIN {X -90.316,Y 3.3389,Z 94,A 172.6479,B 24.92,C -2.065,E1 24.8399,E2 -87.5437} C_DIS
LIN {X -90.1325,Y 6.6531,Z 94,A 170.5242,B 24.9196,C -2.0712,E1 24.8403,E2 -85.422} C_DIS
LIN {X -89.9426,Y 8.858,Z 94,A 169.1085,B 24.9192,C -2.0753,E1 24.8407,E2 -84.0077} C_DIS
LIN {X -89.5566,Y 12.155,Z 94,A 166.9904,B 24.9187,C -2.0816,E1 24.8414,E2 -81.8921} C_DIS
LIN {X -89.0475,Y 15.4492,Z 94,A 164.8605,B 24.9182,C -2.0879,E1 24.8423,E2 -79.7644} C_DIS
LIN {X -88.5347,Y 18.1504,Z 94,A 163.0307,B 24.918,C -2.0909,E1 24.8433,E2 -77.931} C_DIS
LIN {X -87.8673,Y 21.1483,Z 94,A 160.9872,B 24.9177,C -2.0943,E1 24.8446,E2 -75.8836} C_DIS
LIN {X -87.1776,Y 23.8322,Z 94,A 159.3754,B 24.917,C -2.104,E1 24.8457,E2 -74.2857} C_DIS
LIN {X -86.4897,Y 26.2231,Z 94,A 157.662,B 24.917,C -2.105,E1 24.8471,E2 -72.5646} C_DIS
LIN {X -85.5563,Y 29.1209,Z 94,A 155.6683,B 24.9166,C -2.1091,E1 24.8488,E2 -70.5694} C_DIS
LIN {X -84.4139,Y 32.2834,Z 94,A 153.6614,B 24.9158,C -2.1193,E1 24.8508,E2 -68.5756} C_DIS
LIN {X -83.1719,Y 35.3603,Z 94,A 151.5796,B 24.9152,C -2.1264,E1 24.853,E2 -66.4989} C_DIS
LIN {X -82.1685,Y 37.636,Z 94,A 149.8638,B 24.9152,C -2.127,E1 24.855,E2 -64.7753} C_DIS
LIN {X -80.7769,Y 40.5354,Z 94,A 147.767,B 24.9148,C -2.1313,E1 24.8575,E2 -62.6775} C_DIS
LIN {X -79.28,Y 43.3892,Z 94,A 145.8429,B 24.914,C -2.1408,E1 24.86,E2 -60.7658} C_DIS
LIN {X -78.0743,Y 45.525,Z 94,A 144.1055,B 24.9141,C -2.1399,E1 24.8625,E2 -59.0172} C_DIS
LIN {X -76.3696,Y 48.3301,Z 94,A 142.2244,B 24.9132,C -2.1517,E1 24.8652,E2 -57.1545} C_DIS
LIN {X -75.1441,Y 50.2145,Z 94,A 140.7914,B 24.9129,C -2.1554,E1 24.8674,E2 -55.7232} C_DIS
LIN {X -73.8913,Y 52.0405,Z 94,A 139.378,B 24.9126,C -2.159,E1 24.8697,E2 -54.3114} C_DIS
LIN {X -72.5936,Y 53.836,Z 94,A 137.7534,B 24.9128,C -2.1562,E1 24.8724,E2 -52.6724} C_DIS
LIN {X -70.555,Y 56.4811,Z 94,A 135.6195,B 24.9124,C -2.1613,E1 24.8761,E2 -50.5406} C_DIS
LIN {X -68.4325,Y 59.035,Z 94,A 133.5005,B 24.912,C -2.1663,E1 24.8799,E2 -48.4238} C_DIS
LIN {X -66.2174,Y 61.5093,Z 94,A 131.3828,B 24.9116,C -2.1712,E1 24.8839,E2 -46.3085} C_DIS
LIN {X -63.8991,Y 63.9143,Z 94,A 129.2559,B 24.9112,C -2.1761,E1 24.888,E2 -44.1841} C_DIS
Enddeposition()
END
